LIN {X -0.110,Y -591.077,Z 1525.096,A 0.000,B 0.000,C 90.000,E1 53.336} C_DIS
LIN {X 0.114,Y -591.584,Z 1525.089,A 0.000,B 0.000,C 90.000,E1 51.984} C_DIS
LIN {X 0.039,Y -592.394,Z 1525.077,A 0.000,B 0.000,C 90.000,E1 49.865} C_DIS
LIN {X -0.237,Y -592.697,Z 1525.073,A 0.000,B 0.000,C 90.000,E1 49.094} C_DIS
LIN {X 0.093,Y -592.919,Z 1525.067,A 0.000,B 0.000,C 90.000,E1 48.000} C_DIS
LIN {X 0.028,Y -592.937,Z 1525.061,A 0.000,B 0.000,C 90.000,E1 46.944} C_DIS
LIN {X -0.066,Y -592.710,Z 1525.055,A 0.000,B 0.000,C 90.000,E1 45.891} C_DIS
LIN {X -0.158,Y -592.347,Z 1525.049,A 0.000,B 0.000,C 90.000,E1 44.838} C_DIS
LIN {X -0.256,Y -591.689,Z 1525.043,A 0.000,B 0.000,C 90.000,E1 43.785} C_DIS
LIN {X 0.062,Y -590.876,Z 1525.037,A 0.000,B 0.000,C 90.000,E1 42.690} C_DIS
LIN {X 0.018,Y -590.208,Z 1525.034,A 0.000,B 0.000,C 90.000,E1 42.162} C_DIS
LIN {X -0.026,Y -589.196,Z 1525.031,A 0.000,B 0.000,C 90.000,E1 41.634} C_DIS
LIN {X 0.310,Y -587.829,Z 1525.028,A 0.000,B 0.000,C 90.000,E1 41.067} C_DIS
LIN {X 0.059,Y -587.019,Z 1525.027,A 0.000,B 0.000,C 90.000,E1 40.825} C_DIS
LIN {X -0.293,Y -585.430,Z 1525.025,A 0.000,B 0.000,C 90.000,E1 40.458} C_DIS
LIN {X -0.107,Y -583.916,Z 1525.023,A 0.000,B 0.000,C 90.000,E1 40.172} C_DIS
LIN {X -0.139,Y -582.504,Z 1525.022,A 0.000,B 0.000,C 90.000,E1 40.011} C_DIS
LIN {X -0.060,Y -581.396,Z 1525.022,A 0.000,B 0.000,C 90.000,E1 39.930} C_DIS
LIN {X -0.252,Y -580.763,Z 1525.022,A 0.000,B 0.000,C 90.000,E1 39.930} C_DIS
LIN {X 0.106,Y -408.220,Z 1525.022,A 0.000,B 0.000,C 90.000,E1 39.886} C_DIS
LIN {X -0.052,Y -405.621,Z 1525.013,A 0.000,B 0.000,C 90.000,E1 38.382} C_DIS
LIN {X 0.011,Y -396.780,Z 1524.988,A 0.000,B 0.000,C 90.000,E1 33.833} C_DIS
LIN {X -0.015,Y -393.578,Z 1524.976,A 0.000,B 0.000,C 90.000,E1 31.720} C_DIS
LIN {X -0.106,Y -386.207,Z 1524.953,A 0.000,B 0.000,C 90.000,E1 27.462} C_DIS
LIN {X -0.128,Y -382.999,Z 1524.939,A 0.000,B 0.000,C 90.000,E1 24.951} C_DIS
LIN {X -0.025,Y -380.145,Z 1524.929,A 0.000,B 0.000,C 90.000,E1 23.131} C_DIS
LIN {X -0.152,Y -374.085,Z 1524.900,A 0.000,B 0.000,C 90.000,E1 18.055} C_DIS
LIN {X 0.155,Y -373.383,Z 1524.896,A 0.000,B 0.000,C 90.000,E1 17.275} C_DIS
LIN {X 0.170,Y -367.880,Z 1524.868,A 0.000,B 0.000,C 90.000,E1 12.119} C_DIS
LIN {X 0.114,Y -366.486,Z 1524.855,A 0.000,B 0.000,C 90.000,E1 9.905} C_DIS
LIN {X 0.050,Y -361.788,Z 1524.822,A 0.000,B 0.000,C 90.000,E1 3.955} C_DIS
LIN {X -0.065,Y -360.902,Z 1524.801,A 0.000,B 0.000,C 90.000,E1 0.229} C_DIS
LIN {X -0.053,Y -359.426,Z 1524.770,A 0.000,B 0.000,C 90.000,E1 354.546} C_DIS
LIN {X 0.070,Y -358.890,Z 1524.759,A 0.000,B 0.000,C 90.000,E1 352.648} C_DIS
LIN {X -0.020,Y -359.563,Z 1524.726,A 0.000,B 0.000,C 90.000,E1 346.645} C_DIS
LIN {X 0.001,Y -361.801,Z 1524.684,A 0.000,B 0.000,C 90.000,E1 339.135} C_DIS
LIN {X -0.154,Y -362.053,Z 1524.680,A 0.000,B 0.000,C 90.000,E1 338.411} C_DIS
LIN {X 0.189,Y -365.980,Z 1524.643,A 0.000,B 0.000,C 90.000,E1 331.641} C_DIS
LIN {X 0.029,Y -366.387,Z 1524.639,A 0.000,B 0.000,C 90.000,E1 330.923} C_DIS
LIN {X -0.031,Y -371.355,Z 1524.604,A 0.000,B 0.000,C 90.000,E1 324.642} C_DIS
LIN {X -0.043,Y -371.766,Z 1524.602,A 0.000,B 0.000,C 90.000,E1 324.276} C_DIS
LIN {X 0.013,Y -377.358,Z 1524.567,A 0.000,B 0.000,C 90.000,E1 318.038} C_DIS
LIN {X 0.012,Y -378.235,Z 1524.563,A 0.000,B 0.000,C 90.000,E1 317.310} C_DIS
LIN {X 0.002,Y -383.940,Z 1524.531,A 0.000,B 0.000,C 90.000,E1 311.515} C_DIS
LIN {X 0.088,Y -384.893,Z 1524.527,A 0.000,B 0.000,C 90.000,E1 310.782} C_DIS
LIN {X 0.262,Y -390.610,Z 1524.495,A 0.000,B 0.000,C 90.000,E1 305.025} C_DIS
LIN {X 0.106,Y -391.104,Z 1524.493,A 0.000,B 0.000,C 90.000,E1 304.692} C_DIS
LIN {X 0.022,Y -391.648,Z 1524.489,A 0.000,B 0.000,C 90.000,E1 303.992} C_DIS
LIN {X -0.080,Y -396.825,Z 1524.459,A 0.000,B 0.000,C 90.000,E1 298.693} C_DIS
LIN {X -0.210,Y -397.120,Z 1524.457,A 0.000,B 0.000,C 90.000,E1 298.359} C_DIS
LIN {X -0.055,Y -401.597,Z 1524.426,A 0.000,B 0.000,C 90.000,E1 292.717} C_DIS
LIN {X 0.222,Y -404.659,Z 1524.395,A 0.000,B 0.000,C 90.000,E1 287.094} C_DIS
LIN {X -0.079,Y -404.735,Z 1524.391,A 0.000,B 0.000,C 90.000,E1 286.441} C_DIS
LIN {X 0.214,Y -406.099,Z 1524.364,A 0.000,B 0.000,C 90.000,E1 281.535} C_DIS
LIN {X -0.176,Y -406.094,Z 1524.362,A 0.000,B 0.000,C 90.000,E1 281.243} C_DIS
LIN {X -0.097,Y -405.680,Z 1524.333,A 0.000,B 0.000,C 90.000,E1 276.024} C_DIS
LIN {X -0.165,Y -405.058,Z 1524.328,A 0.000,B 0.000,C 90.000,E1 274.992} C_DIS
LIN {X -0.060,Y -403.497,Z 1524.304,A 0.000,B 0.000,C 90.000,E1 270.802} C_DIS
LIN {X -0.092,Y -403.288,Z 1524.302,A 0.000,B 0.000,C 90.000,E1 270.458} C_DIS
LIN {X 0.091,Y -398.931,Z 1524.271,A 0.000,B 0.000,C 90.000,E1 264.837} C_DIS
LIN {X -0.040,Y -393.108,Z 1524.242,A 0.000,B 0.000,C 90.000,E1 259.567} C_DIS
LIN {X -0.079,Y -392.835,Z 1524.240,A 0.000,B 0.000,C 90.000,E1 259.218} C_DIS
LIN {X 0.034,Y -385.993,Z 1524.212,A 0.000,B 0.000,C 90.000,E1 254.212} C_DIS
LIN {X -0.026,Y -385.267,Z 1524.208,A 0.000,B 0.000,C 90.000,E1 253.504} C_DIS
LIN {X -0.004,Y -384.768,Z 1524.206,A 0.000,B 0.000,C 90.000,E1 253.142} C_DIS
LIN {X 0.221,Y -377.973,Z 1524.182,A 0.000,B 0.000,C 90.000,E1 248.773} C_DIS
LIN {X -0.044,Y -376.233,Z 1524.174,A 0.000,B 0.000,C 90.000,E1 247.358} C_DIS
LIN {X 0.057,Y -374.944,Z 1524.170,A 0.000,B 0.000,C 90.000,E1 246.613} C_DIS
LIN {X -0.208,Y -368.417,Z 1524.148,A 0.000,B 0.000,C 90.000,E1 242.615} C_DIS
LIN {X 0.097,Y -366.047,Z 1524.137,A 0.000,B 0.000,C 90.000,E1 240.717} C_DIS
LIN {X 0.004,Y -359.196,Z 1524.115,A 0.000,B 0.000,C 90.000,E1 236.628} C_DIS
LIN {X 0.021,Y -355.842,Z 1524.100,A 0.000,B 0.000,C 90.000,E1 233.989} C_DIS
LIN {X -0.173,Y -348.793,Z 1524.075,A 0.000,B 0.000,C 90.000,E1 229.461} C_DIS
LIN {X -0.097,Y -346.185,Z 1524.062,A 0.000,B 0.000,C 90.000,E1 227.148} C_DIS
LIN {X -0.088,Y -345.065,Z 1524.058,A 0.000,B 0.000,C 90.000,E1 226.377} C_DIS
LIN {X 0.094,Y -338.586,Z 1524.030,A 0.000,B 0.000,C 90.000,E1 221.310} C_DIS
LIN {X 0.094,Y -336.840,Z 1524.019,A 0.000,B 0.000,C 90.000,E1 219.358} C_DIS
LIN {X 0.014,Y -330.861,Z 1523.988,A 0.000,B 0.000,C 90.000,E1 213.865} C_DIS
LIN {X 0.149,Y -329.296,Z 1523.975,A 0.000,B 0.000,C 90.000,E1 211.465} C_DIS
LIN {X -0.154,Y -324.669,Z 1523.942,A 0.000,B 0.000,C 90.000,E1 205.540} C_DIS
LIN {X 0.174,Y -323.837,Z 1523.928,A 0.000,B 0.000,C 90.000,E1 203.078} C_DIS
LIN {X -0.017,Y -321.124,Z 1523.881,A 0.000,B 0.000,C 90.000,E1 194.662} C_DIS
LIN {X 0.138,Y -320.932,Z 1523.877,A 0.000,B 0.000,C 90.000,E1 193.828} C_DIS
LIN {X -0.076,Y -321.562,Z 1523.832,A 0.000,B 0.000,C 90.000,E1 185.796} C_DIS
LIN {X -0.143,Y -324.415,Z 1523.790,A 0.000,B 0.000,C 90.000,E1 178.165} C_DIS
LIN {X -0.141,Y -325.376,Z 1523.783,A 0.000,B 0.000,C 90.000,E1 176.963} C_DIS
LIN {X -0.100,Y -329.112,Z 1523.750,A 0.000,B 0.000,C 90.000,E1 170.971} C_DIS
LIN {X 0.061,Y -334.260,Z 1523.726,A 0.000,B 0.000,C 90.000,E1 166.589} C_DIS
LIN {X 0.067,Y -335.488,Z 1523.719,A 0.000,B 0.000,C 90.000,E1 165.408} C_DIS
LIN {X 0.143,Y -340.932,Z 1523.695,A 0.000,B 0.000,C 90.000,E1 161.094} C_DIS
LIN {X -0.172,Y -342.138,Z 1523.691,A 0.000,B 0.000,C 90.000,E1 160.369} C_DIS
LIN {X -0.058,Y -347.939,Z 1523.667,A 0.000,B 0.000,C 90.000,E1 156.102} C_DIS
LIN {X -0.081,Y -354.259,Z 1523.648,A 0.000,B 0.000,C 90.000,E1 152.666} C_DIS
LIN {X -0.222,Y -361.406,Z 1523.625,A 0.000,B 0.000,C 90.000,E1 148.535} C_DIS
LIN {X 0.065,Y -368.758,Z 1523.606,A 0.000,B 0.000,C 90.000,E1 145.135} C_DIS
LIN {X 0.065,Y -377.029,Z 1523.584,A 0.000,B 0.000,C 90.000,E1 141.090} C_DIS
LIN {X -0.061,Y -383.435,Z 1523.570,A 0.000,B 0.000,C 90.000,E1 138.566} C_DIS
LIN {X -0.015,Y -385.037,Z 1523.566,A 0.000,B 0.000,C 90.000,E1 137.838} C_DIS
LIN {X -0.132,Y -386.364,Z 1523.562,A 0.000,B 0.000,C 90.000,E1 137.229} C_DIS
LIN {X -0.232,Y -540.923,Z 1523.562,A 0.000,B 0.000,C 90.000,E1 137.229} C_DIS
LIN {X 0.102,Y -542.616,Z 1523.562,A 0.000,B 0.000,C 90.000,E1 137.106} C_DIS
LIN {X -0.112,Y -544.188,Z 1523.561,A 0.000,B 0.000,C 90.000,E1 136.944} C_DIS
LIN {X -0.124,Y -545.786,Z 1523.559,A 0.000,B 0.000,C 90.000,E1 136.662} C_DIS
LIN {X -0.104,Y -546.970,Z 1523.558,A 0.000,B 0.000,C 90.000,E1 136.377} C_DIS
LIN {X -0.074,Y -548.801,Z 1523.555,A 0.000,B 0.000,C 90.000,E1 135.810} C_DIS
LIN {X -0.029,Y -550.156,Z 1523.551,A 0.000,B 0.000,C 90.000,E1 135.243} C_DIS
LIN {X 0.028,Y -551.193,Z 1523.548,A 0.000,B 0.000,C 90.000,E1 134.676} C_DIS
LIN {X -0.264,Y -552.360,Z 1523.544,A 0.000,B 0.000,C 90.000,E1 133.866} C_DIS
LIN {X -0.070,Y -553.654,Z 1523.536,A 0.000,B 0.000,C 90.000,E1 132.447} C_DIS
LIN {X -0.227,Y -554.854,Z 1523.528,A 0.000,B 0.000,C 90.000,E1 131.067} C_DIS
LIN {X 0.058,Y -555.934,Z 1523.520,A 0.000,B 0.000,C 90.000,E1 129.644} C_DIS
LIN {X 0.012,Y -556.872,Z 1523.513,A 0.000,B 0.000,C 90.000,E1 128.257} C_DIS
LIN {X -0.017,Y -557.730,Z 1523.505,A 0.000,B 0.000,C 90.000,E1 126.870} C_DIS
LIN {X 0.321,Y -558.307,Z 1523.499,A 0.000,B 0.000,C 90.000,E1 125.724} C_DIS
LIN {X -0.117,Y -558.754,Z 1523.493,A 0.000,B 0.000,C 90.000,E1 124.659} C_DIS
LIN {X 0.370,Y -559.049,Z 1523.486,A 0.000,B 0.000,C 90.000,E1 123.499} C_DIS
LIN {X 0.176,Y -559.194,Z 1523.479,A 0.000,B 0.000,C 90.000,E1 122.133} C_DIS
LIN {X -0.106,Y -559.571,Z 1523.465,A 0.000,B 0.000,C 90.000,E1 119.667} C_DIS
LIN {X -0.106,Y -559.896,Z 1523.457,A 0.000,B 0.000,C 90.000,E1 118.281} C_DIS
LIN {X 0.128,Y -560.256,Z 1523.449,A 0.000,B 0.000,C 90.000,E1 116.873} C_DIS
LIN {X -0.133,Y -560.520,Z 1523.442,A 0.000,B 0.000,C 90.000,E1 115.515} C_DIS
LIN {X -0.027,Y -560.874,Z 1523.431,A 0.000,B 0.000,C 90.000,E1 113.567} C_DIS
LIN {X -0.240,Y -561.086,Z 1523.423,A 0.000,B 0.000,C 90.000,E1 112.206} C_DIS
LIN {X 0.075,Y -561.325,Z 1523.416,A 0.000,B 0.000,C 90.000,E1 110.791} C_DIS
LIN {X -0.016,Y -561.627,Z 1523.406,A 0.000,B 0.000,C 90.000,E1 109.141} C_DIS
LIN {X 0.246,Y -561.910,Z 1523.397,A 0.000,B 0.000,C 90.000,E1 107.457} C_DIS
LIN {X -0.185,Y -562.229,Z 1523.388,A 0.000,B 0.000,C 90.000,E1 105.843} C_DIS
LIN {X -0.074,Y -562.589,Z 1523.379,A 0.000,B 0.000,C 90.000,E1 104.175} C_DIS
LIN {X -0.229,Y -563.011,Z 1523.370,A 0.000,B 0.000,C 90.000,E1 102.535} C_DIS
LIN {X -0.206,Y -563.703,Z 1523.359,A 0.000,B 0.000,C 90.000,E1 100.602} C_DIS
LIN {X 0.276,Y -564.452,Z 1523.348,A 0.000,B 0.000,C 90.000,E1 98.624} C_DIS
LIN {X -0.196,Y -565.016,Z 1523.340,A 0.000,B 0.000,C 90.000,E1 97.296} C_DIS
LIN {X 0.001,Y -565.710,Z 1523.331,A 0.000,B 0.000,C 90.000,E1 95.625} C_DIS
LIN {X -0.246,Y -566.525,Z 1523.321,A 0.000,B 0.000,C 90.000,E1 93.726} C_DIS
LIN {X -0.095,Y -567.254,Z 1523.311,A 0.000,B 0.000,C 90.000,E1 92.064} C_DIS
LIN {X -0.048,Y -567.928,Z 1523.304,A 0.000,B 0.000,C 90.000,E1 90.688} C_DIS
LIN {X 0.123,Y -568.719,Z 1523.295,A 0.000,B 0.000,C 90.000,E1 89.026} C_DIS
LIN {X 0.031,Y -569.821,Z 1523.283,A 0.000,B 0.000,C 90.000,E1 86.846} C_DIS
LIN {X -0.154,Y -570.797,Z 1523.272,A 0.000,B 0.000,C 90.000,E1 84.951} C_DIS
LIN {X -0.011,Y -571.595,Z 1523.264,A 0.000,B 0.000,C 90.000,E1 83.571} C_DIS
LIN {X 0.022,Y -572.832,Z 1523.254,A 0.000,B 0.000,C 90.000,E1 81.659} C_DIS
LIN {X 0.092,Y -574.108,Z 1523.243,A 0.000,B 0.000,C 90.000,E1 79.746} C_DIS
LIN {X -0.283,Y -575.573,Z 1523.233,A 0.000,B 0.000,C 90.000,E1 77.881} C_DIS
LIN {X -0.026,Y -576.844,Z 1523.224,A 0.000,B 0.000,C 90.000,E1 76.228} C_DIS
LIN {X -0.307,Y -577.653,Z 1523.218,A 0.000,B 0.000,C 90.000,E1 75.172} C_DIS
LIN {X -0.205,Y -578.921,Z 1523.207,A 0.000,B 0.000,C 90.000,E1 73.268} C_DIS
LIN {X -0.075,Y -580.324,Z 1523.195,A 0.000,B 0.000,C 90.000,E1 71.094} C_DIS
LIN {X -0.190,Y -580.822,Z 1523.190,A 0.000,B 0.000,C 90.000,E1 70.296} C_DIS
LIN {X 0.147,Y -581.736,Z 1523.182,A 0.000,B 0.000,C 90.000,E1 68.646} C_DIS
LIN {X -0.185,Y -582.761,Z 1523.171,A 0.000,B 0.000,C 90.000,E1 66.794} C_DIS
LIN {X -0.274,Y -583.826,Z 1523.161,A 0.000,B 0.000,C 90.000,E1 64.921} C_DIS
LIN {X -0.213,Y -585.515,Z 1523.146,A 0.000,B 0.000,C 90.000,E1 62.231} C_DIS
LIN {X 0.137,Y -586.676,Z 1523.137,A 0.000,B 0.000,C 90.000,E1 60.589} C_DIS
LIN {X -0.175,Y -587.630,Z 1523.129,A 0.000,B 0.000,C 90.000,E1 59.282} C_DIS
LIN {X 0.134,Y -588.545,Z 1523.122,A 0.000,B 0.000,C 90.000,E1 57.916} C_DIS
LIN {X 0.146,Y -589.451,Z 1523.115,A 0.000,B 0.000,C 90.000,E1 56.580} C_DIS
LIN {X -0.003,Y -590.403,Z 1523.107,A 0.000,B 0.000,C 90.000,E1 55.261} C_DIS
LIN {X -0.199,Y -591.398,Z 1523.097,A 0.000,B 0.000,C 90.000,E1 53.417} C_DIS
LIN {X 0.028,Y -591.926,Z 1523.089,A 0.000,B 0.000,C 90.000,E1 52.065} C_DIS
LIN {X 0.342,Y -592.766,Z 1523.078,A 0.000,B 0.000,C 90.000,E1 49.908} C_DIS
LIN {X 0.283,Y -593.108,Z 1523.072,A 0.000,B 0.000,C 90.000,E1 48.852} C_DIS
LIN {X 0.020,Y -593.337,Z 1523.067,A 0.000,B 0.000,C 90.000,E1 48.081} C_DIS
LIN {X -0.039,Y -593.355,Z 1523.061,A 0.000,B 0.000,C 90.000,E1 47.025} C_DIS
LIN {X -0.359,Y -593.143,Z 1523.054,A 0.000,B 0.000,C 90.000,E1 45.729} C_DIS
LIN {X -0.029,Y -592.727,Z 1523.048,A 0.000,B 0.000,C 90.000,E1 44.636} C_DIS
LIN {X 0.061,Y -591.812,Z 1523.041,A 0.000,B 0.000,C 90.000,E1 43.299} C_DIS
LIN {X -0.019,Y -590.948,Z 1523.035,A 0.000,B 0.000,C 90.000,E1 42.243} C_DIS
LIN {X 0.090,Y -589.887,Z 1523.030,A 0.000,B 0.000,C 90.000,E1 41.434} C_DIS
LIN {X 0.040,Y -588.904,Z 1523.027,A 0.000,B 0.000,C 90.000,E1 40.906} C_DIS
LIN {X -0.016,Y -587.630,Z 1523.024,A 0.000,B 0.000,C 90.000,E1 40.378} C_DIS
LIN {X 0.177,Y -586.831,Z 1523.023,A 0.000,B 0.000,C 90.000,E1 40.092} C_DIS
LIN {X -0.080,Y -585.891,Z 1523.021,A 0.000,B 0.000,C 90.000,E1 39.850} C_DIS
LIN {X 0.109,Y -584.616,Z 1523.020,A 0.000,B 0.000,C 90.000,E1 39.564} C_DIS
LIN {X 0.016,Y -583.816,Z 1523.019,A 0.000,B 0.000,C 90.000,E1 39.439} C_DIS
LIN {X -0.294,Y -582.284,Z 1523.018,A 0.000,B 0.000,C 90.000,E1 39.277} C_DIS
LIN {X -0.299,Y -581.245,Z 1523.018,A 0.000,B 0.000,C 90.000,E1 39.197} C_DIS
LIN {X 0.095,Y -580.125,Z 1523.017,A 0.000,B 0.000,C 90.000,E1 39.116} C_DIS
LIN {X 0.043,Y -406.894,Z 1523.017,A 0.000,B 0.000,C 90.000,E1 39.116} C_DIS
LIN {X 0.050,Y -405.552,Z 1523.013,A 0.000,B 0.000,C 90.000,E1 38.338} C_DIS
LIN {X 0.125,Y -396.729,Z 1522.988,A 0.000,B 0.000,C 90.000,E1 33.785} C_DIS
LIN {X 0.105,Y -393.515,Z 1522.976,A 0.000,B 0.000,C 90.000,E1 31.671} C_DIS
LIN {X 0.200,Y -386.161,Z 1522.952,A 0.000,B 0.000,C 90.000,E1 27.385} C_DIS
LIN {X 0.006,Y -382.963,Z 1522.938,A 0.000,B 0.000,C 90.000,E1 24.899} C_DIS
LIN {X 0.104,Y -376.256,Z 1522.912,A 0.000,B 0.000,C 90.000,E1 20.174} C_DIS
LIN {X -0.031,Y -373.747,Z 1522.898,A 0.000,B 0.000,C 90.000,E1 17.638} C_DIS
LIN {X -0.112,Y -372.359,Z 1522.892,A 0.000,B 0.000,C 90.000,E1 16.551} C_DIS
LIN {X -0.030,Y -367.091,Z 1522.861,A 0.000,B 0.000,C 90.000,E1 11.007} C_DIS
LIN {X -0.096,Y -366.466,Z 1522.855,A 0.000,B 0.000,C 90.000,E1 9.905} C_DIS
LIN {X -0.158,Y -361.773,Z 1522.822,A 0.000,B 0.000,C 90.000,E1 3.955} C_DIS
LIN {X 0.088,Y -360.895,Z 1522.801,A 0.000,B 0.000,C 90.000,E1 0.172} C_DIS
LIN {X -0.053,Y -359.426,Z 1522.770,A 0.000,B 0.000,C 90.000,E1 354.546} C_DIS
LIN {X 0.070,Y -358.890,Z 1522.759,A 0.000,B 0.000,C 90.000,E1 352.648} C_DIS
LIN {X -0.020,Y -359.563,Z 1522.726,A 0.000,B 0.000,C 90.000,E1 346.645} C_DIS
LIN {X 0.001,Y -361.801,Z 1522.684,A 0.000,B 0.000,C 90.000,E1 339.135} C_DIS
LIN {X -0.154,Y -362.053,Z 1522.680,A 0.000,B 0.000,C 90.000,E1 338.411} C_DIS
LIN {X 0.189,Y -365.980,Z 1522.643,A 0.000,B 0.000,C 90.000,E1 331.641} C_DIS
LIN {X 0.029,Y -366.387,Z 1522.639,A 0.000,B 0.000,C 90.000,E1 330.923} C_DIS
LIN {X -0.031,Y -371.355,Z 1522.604,A 0.000,B 0.000,C 90.000,E1 324.642} C_DIS
LIN {X -0.043,Y -371.766,Z 1522.602,A 0.000,B 0.000,C 90.000,E1 324.276} C_DIS
LIN {X 0.013,Y -377.358,Z 1522.567,A 0.000,B 0.000,C 90.000,E1 318.038} C_DIS
LIN {X 0.012,Y -378.235,Z 1522.563,A 0.000,B 0.000,C 90.000,E1 317.310} C_DIS
LIN {X 0.002,Y -383.940,Z 1522.531,A 0.000,B 0.000,C 90.000,E1 311.515} C_DIS
LIN {X 0.088,Y -384.893,Z 1522.527,A 0.000,B 0.000,C 90.000,E1 310.782} C_DIS
LIN {X 0.262,Y -390.610,Z 1522.495,A 0.000,B 0.000,C 90.000,E1 305.025} C_DIS
LIN {X 0.106,Y -391.104,Z 1522.493,A 0.000,B 0.000,C 90.000,E1 304.692} C_DIS
LIN {X 0.022,Y -391.648,Z 1522.489,A 0.000,B 0.000,C 90.000,E1 303.992} C_DIS
LIN {X -0.080,Y -396.825,Z 1522.459,A 0.000,B 0.000,C 90.000,E1 298.693} C_DIS
LIN {X -0.210,Y -397.120,Z 1522.457,A 0.000,B 0.000,C 90.000,E1 298.359} C_DIS
LIN {X -0.055,Y -401.597,Z 1522.426,A 0.000,B 0.000,C 90.000,E1 292.717} C_DIS
LIN {X 0.222,Y -404.659,Z 1522.395,A 0.000,B 0.000,C 90.000,E1 287.094} C_DIS
LIN {X -0.079,Y -404.735,Z 1522.391,A 0.000,B 0.000,C 90.000,E1 286.441} C_DIS
LIN {X 0.214,Y -406.099,Z 1522.364,A 0.000,B 0.000,C 90.000,E1 281.535} C_DIS
LIN {X -0.176,Y -406.094,Z 1522.362,A 0.000,B 0.000,C 90.000,E1 281.243} C_DIS
LIN {X -0.097,Y -405.680,Z 1522.333,A 0.000,B 0.000,C 90.000,E1 276.024} C_DIS
LIN {X -0.165,Y -405.058,Z 1522.328,A 0.000,B 0.000,C 90.000,E1 274.992} C_DIS
LIN {X -0.060,Y -403.497,Z 1522.304,A 0.000,B 0.000,C 90.000,E1 270.802} C_DIS
LIN {X -0.092,Y -403.288,Z 1522.302,A 0.000,B 0.000,C 90.000,E1 270.458} C_DIS
LIN {X 0.091,Y -398.931,Z 1522.271,A 0.000,B 0.000,C 90.000,E1 264.837} C_DIS
LIN {X -0.040,Y -393.108,Z 1522.242,A 0.000,B 0.000,C 90.000,E1 259.567} C_DIS
LIN {X -0.079,Y -392.835,Z 1522.240,A 0.000,B 0.000,C 90.000,E1 259.218} C_DIS
LIN {X 0.034,Y -385.993,Z 1522.212,A 0.000,B 0.000,C 90.000,E1 254.212} C_DIS
LIN {X -0.026,Y -385.267,Z 1522.208,A 0.000,B 0.000,C 90.000,E1 253.504} C_DIS
LIN {X -0.004,Y -384.768,Z 1522.206,A 0.000,B 0.000,C 90.000,E1 253.142} C_DIS
LIN {X 0.221,Y -377.973,Z 1522.182,A 0.000,B 0.000,C 90.000,E1 248.773} C_DIS
LIN {X -0.044,Y -376.233,Z 1522.174,A 0.000,B 0.000,C 90.000,E1 247.358} C_DIS
LIN {X 0.057,Y -374.944,Z 1522.170,A 0.000,B 0.000,C 90.000,E1 246.613} C_DIS
LIN {X -0.208,Y -368.417,Z 1522.148,A 0.000,B 0.000,C 90.000,E1 242.615} C_DIS
LIN {X 0.097,Y -366.047,Z 1522.137,A 0.000,B 0.000,C 90.000,E1 240.717} C_DIS
LIN {X 0.004,Y -359.196,Z 1522.115,A 0.000,B 0.000,C 90.000,E1 236.628} C_DIS
LIN {X 0.021,Y -355.842,Z 1522.100,A 0.000,B 0.000,C 90.000,E1 233.989} C_DIS
LIN {X -0.173,Y -348.793,Z 1522.075,A 0.000,B 0.000,C 90.000,E1 229.461} C_DIS
LIN {X -0.097,Y -346.185,Z 1522.062,A 0.000,B 0.000,C 90.000,E1 227.148} C_DIS
LIN {X -0.088,Y -345.065,Z 1522.058,A 0.000,B 0.000,C 90.000,E1 226.377} C_DIS
LIN {X 0.094,Y -338.586,Z 1522.030,A 0.000,B 0.000,C 90.000,E1 221.310} C_DIS
LIN {X 0.094,Y -336.840,Z 1522.019,A 0.000,B 0.000,C 90.000,E1 219.358} C_DIS
LIN {X 0.014,Y -330.861,Z 1521.988,A 0.000,B 0.000,C 90.000,E1 213.865} C_DIS
LIN {X 0.149,Y -329.296,Z 1521.975,A 0.000,B 0.000,C 90.000,E1 211.465} C_DIS
LIN {X -0.154,Y -324.669,Z 1521.942,A 0.000,B 0.000,C 90.000,E1 205.540} C_DIS
LIN {X 0.174,Y -323.837,Z 1521.928,A 0.000,B 0.000,C 90.000,E1 203.078} C_DIS
LIN {X -0.017,Y -321.124,Z 1521.881,A 0.000,B 0.000,C 90.000,E1 194.662} C_DIS
LIN {X 0.138,Y -320.932,Z 1521.877,A 0.000,B 0.000,C 90.000,E1 193.828} C_DIS
LIN {X -0.076,Y -321.562,Z 1521.832,A 0.000,B 0.000,C 90.000,E1 185.796} C_DIS
LIN {X -0.143,Y -324.415,Z 1521.790,A 0.000,B 0.000,C 90.000,E1 178.165} C_DIS
LIN {X -0.141,Y -325.376,Z 1521.783,A 0.000,B 0.000,C 90.000,E1 176.963} C_DIS
LIN {X -0.100,Y -329.112,Z 1521.750,A 0.000,B 0.000,C 90.000,E1 170.971} C_DIS
LIN {X 0.061,Y -334.260,Z 1521.726,A 0.000,B 0.000,C 90.000,E1 166.589} C_DIS
LIN {X 0.067,Y -335.488,Z 1521.719,A 0.000,B 0.000,C 90.000,E1 165.408} C_DIS
LIN {X 0.143,Y -340.932,Z 1521.695,A 0.000,B 0.000,C 90.000,E1 161.094} C_DIS
LIN {X -0.172,Y -342.138,Z 1521.691,A 0.000,B 0.000,C 90.000,E1 160.369} C_DIS
LIN {X -0.058,Y -347.939,Z 1521.667,A 0.000,B 0.000,C 90.000,E1 156.102} C_DIS
LIN {X -0.081,Y -354.259,Z 1521.648,A 0.000,B 0.000,C 90.000,E1 152.666} C_DIS
LIN {X -0.222,Y -361.406,Z 1521.625,A 0.000,B 0.000,C 90.000,E1 148.535} C_DIS
LIN {X 0.065,Y -368.758,Z 1521.606,A 0.000,B 0.000,C 90.000,E1 145.135} C_DIS
LIN {X 0.065,Y -377.029,Z 1521.584,A 0.000,B 0.000,C 90.000,E1 141.090} C_DIS
LIN {X -0.061,Y -383.435,Z 1521.570,A 0.000,B 0.000,C 90.000,E1 138.566} C_DIS
LIN {X -0.153,Y -384.579,Z 1521.567,A 0.000,B 0.000,C 90.000,E1 138.081} C_DIS
LIN {X -0.249,Y -540.182,Z 1521.567,A 0.000,B 0.000,C 90.000,E1 138.081} C_DIS
LIN {X 0.231,Y -542.118,Z 1521.566,A 0.000,B 0.000,C 90.000,E1 137.919} C_DIS
LIN {X -0.021,Y -543.063,Z 1521.566,A 0.000,B 0.000,C 90.000,E1 137.838} C_DIS
LIN {X -0.196,Y -544.018,Z 1521.565,A 0.000,B 0.000,C 90.000,E1 137.715} C_DIS
LIN {X 0.190,Y -545.485,Z 1521.563,A 0.000,B 0.000,C 90.000,E1 137.391} C_DIS
LIN {X 0.010,Y -547.099,Z 1521.561,A 0.000,B 0.000,C 90.000,E1 136.986} C_DIS
LIN {X 0.042,Y -548.741,Z 1521.558,A 0.000,B 0.000,C 90.000,E1 136.419} C_DIS
LIN {X -0.293,Y -550.004,Z 1521.555,A 0.000,B 0.000,C 90.000,E1 135.891} C_DIS
LIN {X -0.239,Y -550.989,Z 1521.552,A 0.000,B 0.000,C 90.000,E1 135.324} C_DIS
LIN {X 0.248,Y -552.037,Z 1521.547,A 0.000,B 0.000,C 90.000,E1 134.433} C_DIS
LIN {X -0.035,Y -552.923,Z 1521.542,A 0.000,B 0.000,C 90.000,E1 133.623} C_DIS
LIN {X 0.168,Y -554.208,Z 1521.535,A 0.000,B 0.000,C 90.000,E1 132.204} C_DIS
LIN {X 0.017,Y -555.349,Z 1521.527,A 0.000,B 0.000,C 90.000,E1 130.825} C_DIS
LIN {X -0.122,Y -556.209,Z 1521.521,A 0.000,B 0.000,C 90.000,E1 129.725} C_DIS
LIN {X 0.265,Y -557.294,Z 1521.511,A 0.000,B 0.000,C 90.000,E1 128.016} C_DIS
LIN {X -0.099,Y -558.114,Z 1521.504,A 0.000,B 0.000,C 90.000,E1 126.664} C_DIS
LIN {X 0.247,Y -558.649,Z 1521.498,A 0.000,B 0.000,C 90.000,E1 125.518} C_DIS
LIN {X 0.360,Y -559.144,Z 1521.490,A 0.000,B 0.000,C 90.000,E1 124.119} C_DIS
LIN {X 0.083,Y -559.329,Z 1521.484,A 0.000,B 0.000,C 90.000,E1 123.038} C_DIS
LIN {X -0.102,Y -559.376,Z 1521.476,A 0.000,B 0.000,C 90.000,E1 121.671} C_DIS
LIN {X 0.115,Y -559.816,Z 1521.462,A 0.000,B 0.000,C 90.000,E1 119.155} C_DIS
LIN {X -0.081,Y -560.211,Z 1521.453,A 0.000,B 0.000,C 90.000,E1 117.513} C_DIS
LIN {X -0.138,Y -560.473,Z 1521.447,A 0.000,B 0.000,C 90.000,E1 116.411} C_DIS
LIN {X 0.173,Y -560.756,Z 1521.438,A 0.000,B 0.000,C 90.000,E1 114.719} C_DIS
LIN {X -0.014,Y -561.098,Z 1521.428,A 0.000,B 0.000,C 90.000,E1 113.078} C_DIS
LIN {X -0.114,Y -561.421,Z 1521.417,A 0.000,B 0.000,C 90.000,E1 111.153} C_DIS
LIN {X -0.081,Y -561.731,Z 1521.407,A 0.000,B 0.000,C 90.000,E1 109.214} C_DIS
LIN {X -0.342,Y -562.018,Z 1521.398,A 0.000,B 0.000,C 90.000,E1 107.583} C_DIS
LIN {X -0.070,Y -562.339,Z 1521.388,A 0.000,B 0.000,C 90.000,E1 105.898} C_DIS
LIN {X -0.254,Y -562.667,Z 1521.381,A 0.000,B 0.000,C 90.000,E1 104.537} C_DIS
LIN {X -0.118,Y -563.156,Z 1521.370,A 0.000,B 0.000,C 90.000,E1 102.591} C_DIS
LIN {X 0.066,Y -563.933,Z 1521.358,A 0.000,B 0.000,C 90.000,E1 100.366} C_DIS
LIN {X 0.070,Y -564.861,Z 1521.345,A 0.000,B 0.000,C 90.000,E1 98.163} C_DIS
LIN {X -0.235,Y -565.506,Z 1521.336,A 0.000,B 0.000,C 90.000,E1 96.543} C_DIS
LIN {X -0.190,Y -566.084,Z 1521.329,A 0.000,B 0.000,C 90.000,E1 95.163} C_DIS
LIN {X -0.129,Y -566.724,Z 1521.321,A 0.000,B 0.000,C 90.000,E1 93.784} C_DIS
LIN {X 0.145,Y -567.588,Z 1521.310,A 0.000,B 0.000,C 90.000,E1 91.835} C_DIS
LIN {X 0.199,Y -568.277,Z 1521.303,A 0.000,B 0.000,C 90.000,E1 90.458} C_DIS
LIN {X -0.191,Y -569.093,Z 1521.294,A 0.000,B 0.000,C 90.000,E1 88.854} C_DIS
LIN {X 0.137,Y -570.094,Z 1521.283,A 0.000,B 0.000,C 90.000,E1 86.906} C_DIS
LIN {X -0.010,Y -571.088,Z 1521.272,A 0.000,B 0.000,C 90.000,E1 85.008} C_DIS
LIN {X 0.141,Y -571.885,Z 1521.265,A 0.000,B 0.000,C 90.000,E1 83.628} C_DIS
LIN {X 0.100,Y -573.123,Z 1521.254,A 0.000,B 0.000,C 90.000,E1 81.724} C_DIS
LIN {X 0.264,Y -574.398,Z 1521.244,A 0.000,B 0.000,C 90.000,E1 79.803} C_DIS
LIN {X 0.256,Y -575.625,Z 1521.234,A 0.000,B 0.000,C 90.000,E1 78.173} C_DIS
LIN {X -0.180,Y -576.906,Z 1521.225,A 0.000,B 0.000,C 90.000,E1 76.589} C_DIS
LIN {X -0.107,Y -577.940,Z 1521.218,A 0.000,B 0.000,C 90.000,E1 75.227} C_DIS
LIN {X -0.202,Y -579.007,Z 1521.209,A 0.000,B 0.000,C 90.000,E1 73.614} C_DIS
LIN {X 0.072,Y -579.861,Z 1521.201,A 0.000,B 0.000,C 90.000,E1 72.236} C_DIS
LIN {X -0.154,Y -581.121,Z 1521.191,A 0.000,B 0.000,C 90.000,E1 70.369} C_DIS
LIN {X 0.037,Y -582.156,Z 1521.180,A 0.000,B 0.000,C 90.000,E1 68.465} C_DIS
LIN {X -0.289,Y -583.194,Z 1521.170,A 0.000,B 0.000,C 90.000,E1 66.613} C_DIS
LIN {X -0.127,Y -584.250,Z 1521.160,A 0.000,B 0.000,C 90.000,E1 64.717} C_DIS
LIN {X -0.038,Y -585.986,Z 1521.145,A 0.000,B 0.000,C 90.000,E1 62.025} C_DIS
LIN {X 0.160,Y -586.994,Z 1521.137,A 0.000,B 0.000,C 90.000,E1 60.667} C_DIS
LIN {X 0.029,Y -588.093,Z 1521.128,A 0.000,B 0.000,C 90.000,E1 59.076} C_DIS
LIN {X 0.035,Y -589.004,Z 1521.121,A 0.000,B 0.000,C 90.000,E1 57.740} C_DIS
LIN {X -0.122,Y -589.906,Z 1521.113,A 0.000,B 0.000,C 90.000,E1 56.421} C_DIS
LIN {X -0.256,Y -590.868,Z 1521.106,A 0.000,B 0.000,C 90.000,E1 55.102} C_DIS
LIN {X -0.170,Y -591.696,Z 1521.097,A 0.000,B 0.000,C 90.000,E1 53.497} C_DIS
LIN {X 0.060,Y -592.261,Z 1521.090,A 0.000,B 0.000,C 90.000,E1 52.145} C_DIS
LIN {X -0.047,Y -592.871,Z 1521.081,A 0.000,B 0.000,C 90.000,E1 50.561} C_DIS
LIN {X 0.326,Y -593.519,Z 1521.072,A 0.000,B 0.000,C 90.000,E1 48.933} C_DIS
LIN {X -0.167,Y -593.738,Z 1521.066,A 0.000,B 0.000,C 90.000,E1 47.919} C_DIS
LIN {X 0.186,Y -593.735,Z 1521.060,A 0.000,B 0.000,C 90.000,E1 46.824} C_DIS
LIN {X 0.306,Y -593.535,Z 1521.053,A 0.000,B 0.000,C 90.000,E1 45.486} C_DIS
LIN {X 0.225,Y -593.037,Z 1521.047,A 0.000,B 0.000,C 90.000,E1 44.433} C_DIS
LIN {X 0.134,Y -592.349,Z 1521.041,A 0.000,B 0.000,C 90.000,E1 43.380} C_DIS
LIN {X 0.060,Y -591.464,Z 1521.035,A 0.000,B 0.000,C 90.000,E1 42.324} C_DIS
LIN {X -0.069,Y -590.277,Z 1521.029,A 0.000,B 0.000,C 90.000,E1 41.272} C_DIS
LIN {X -0.117,Y -589.582,Z 1521.026,A 0.000,B 0.000,C 90.000,E1 40.744} C_DIS
LIN {X 0.280,Y -588.642,Z 1521.023,A 0.000,B 0.000,C 90.000,E1 40.172} C_DIS
LIN {X 0.027,Y -588.080,Z 1521.022,A 0.000,B 0.000,C 90.000,E1 39.930} C_DIS
LIN {X 0.224,Y -587.372,Z 1521.020,A 0.000,B 0.000,C 90.000,E1 39.644} C_DIS
LIN {X -0.035,Y -586.521,Z 1521.019,A 0.000,B 0.000,C 90.000,E1 39.402} C_DIS
LIN {X 0.157,Y -585.537,Z 1521.017,A 0.000,B 0.000,C 90.000,E1 39.116} C_DIS
LIN {X 0.346,Y -584.347,Z 1521.016,A 0.000,B 0.000,C 90.000,E1 38.830} C_DIS
LIN {X -0.198,Y -583.596,Z 1521.015,A 0.000,B 0.000,C 90.000,E1 38.749} C_DIS
LIN {X -0.053,Y -582.185,Z 1521.014,A 0.000,B 0.000,C 90.000,E1 38.543} C_DIS
LIN {X -0.345,Y -580.988,Z 1521.014,A 0.000,B 0.000,C 90.000,E1 38.463} C_DIS
LIN {X -0.073,Y -579.954,Z 1521.013,A 0.000,B 0.000,C 90.000,E1 38.382} C_DIS
LIN {X -0.209,Y -579.391,Z 1521.013,A 0.000,B 0.000,C 90.000,E1 38.382} C_DIS
LIN {X -0.170,Y -405.584,Z 1521.013,A 0.000,B 0.000,C 90.000,E1 38.382} C_DIS
LIN {X 0.125,Y -397.278,Z 1520.990,A 0.000,B 0.000,C 90.000,E1 34.119} C_DIS
LIN {X 0.115,Y -394.054,Z 1520.978,A 0.000,B 0.000,C 90.000,E1 32.005} C_DIS
LIN {X -0.019,Y -393.478,Z 1520.976,A 0.000,B 0.000,C 90.000,E1 31.671} C_DIS
LIN {X 0.077,Y -386.135,Z 1520.952,A 0.000,B 0.000,C 90.000,E1 27.385} C_DIS
LIN {X -0.117,Y -382.943,Z 1520.938,A 0.000,B 0.000,C 90.000,E1 24.899} C_DIS
LIN {X -0.018,Y -376.235,Z 1520.912,A 0.000,B 0.000,C 90.000,E1 20.174} C_DIS
LIN {X -0.153,Y -373.731,Z 1520.898,A 0.000,B 0.000,C 90.000,E1 17.638} C_DIS
LIN {X 0.091,Y -371.871,Z 1520.890,A 0.000,B 0.000,C 90.000,E1 16.134} C_DIS
LIN {X 0.068,Y -366.857,Z 1520.859,A 0.000,B 0.000,C 90.000,E1 10.602} C_DIS
LIN {X 0.145,Y -366.452,Z 1520.855,A 0.000,B 0.000,C 90.000,E1 9.849} C_DIS
LIN {X 0.082,Y -361.764,Z 1520.822,A 0.000,B 0.000,C 90.000,E1 3.898} C_DIS
LIN {X -0.033,Y -360.889,Z 1520.801,A 0.000,B 0.000,C 90.000,E1 0.172} C_DIS
LIN {X -0.053,Y -359.426,Z 1520.770,A 0.000,B 0.000,C 90.000,E1 354.546} C_DIS
LIN {X 0.070,Y -358.890,Z 1520.759,A 0.000,B 0.000,C 90.000,E1 352.648} C_DIS
LIN {X -0.020,Y -359.563,Z 1520.726,A 0.000,B 0.000,C 90.000,E1 346.645} C_DIS
LIN {X 0.001,Y -361.801,Z 1520.684,A 0.000,B 0.000,C 90.000,E1 339.135} C_DIS
LIN {X -0.154,Y -362.053,Z 1520.680,A 0.000,B 0.000,C 90.000,E1 338.411} C_DIS
LIN {X 0.189,Y -365.980,Z 1520.643,A 0.000,B 0.000,C 90.000,E1 331.641} C_DIS
LIN {X 0.029,Y -366.387,Z 1520.639,A 0.000,B 0.000,C 90.000,E1 330.923} C_DIS
LIN {X -0.031,Y -371.355,Z 1520.604,A 0.000,B 0.000,C 90.000,E1 324.642} C_DIS
LIN {X -0.043,Y -371.766,Z 1520.602,A 0.000,B 0.000,C 90.000,E1 324.276} C_DIS
LIN {X 0.013,Y -377.358,Z 1520.567,A 0.000,B 0.000,C 90.000,E1 318.038} C_DIS
LIN {X 0.012,Y -378.235,Z 1520.563,A 0.000,B 0.000,C 90.000,E1 317.310} C_DIS
LIN {X 0.002,Y -383.940,Z 1520.531,A 0.000,B 0.000,C 90.000,E1 311.515} C_DIS
LIN {X 0.088,Y -384.893,Z 1520.527,A 0.000,B 0.000,C 90.000,E1 310.782} C_DIS
LIN {X 0.262,Y -390.610,Z 1520.495,A 0.000,B 0.000,C 90.000,E1 305.025} C_DIS
LIN {X 0.106,Y -391.104,Z 1520.493,A 0.000,B 0.000,C 90.000,E1 304.692} C_DIS
LIN {X 0.022,Y -391.648,Z 1520.489,A 0.000,B 0.000,C 90.000,E1 303.992} C_DIS
LIN {X -0.080,Y -396.825,Z 1520.459,A 0.000,B 0.000,C 90.000,E1 298.693} C_DIS
LIN {X -0.210,Y -397.120,Z 1520.457,A 0.000,B 0.000,C 90.000,E1 298.359} C_DIS
LIN {X -0.055,Y -401.597,Z 1520.426,A 0.000,B 0.000,C 90.000,E1 292.717} C_DIS
LIN {X 0.222,Y -404.659,Z 1520.395,A 0.000,B 0.000,C 90.000,E1 287.094} C_DIS
LIN {X -0.079,Y -404.735,Z 1520.391,A 0.000,B 0.000,C 90.000,E1 286.441} C_DIS
LIN {X 0.214,Y -406.099,Z 1520.364,A 0.000,B 0.000,C 90.000,E1 281.535} C_DIS
LIN {X -0.176,Y -406.094,Z 1520.362,A 0.000,B 0.000,C 90.000,E1 281.243} C_DIS
LIN {X -0.097,Y -405.680,Z 1520.333,A 0.000,B 0.000,C 90.000,E1 276.024} C_DIS
LIN {X -0.165,Y -405.058,Z 1520.328,A 0.000,B 0.000,C 90.000,E1 274.992} C_DIS
LIN {X -0.060,Y -403.497,Z 1520.304,A 0.000,B 0.000,C 90.000,E1 270.802} C_DIS
LIN {X -0.092,Y -403.288,Z 1520.302,A 0.000,B 0.000,C 90.000,E1 270.458} C_DIS
LIN {X 0.091,Y -398.931,Z 1520.271,A 0.000,B 0.000,C 90.000,E1 264.837} C_DIS
LIN {X -0.040,Y -393.108,Z 1520.242,A 0.000,B 0.000,C 90.000,E1 259.567} C_DIS
LIN {X -0.079,Y -392.835,Z 1520.240,A 0.000,B 0.000,C 90.000,E1 259.218} C_DIS
LIN {X 0.034,Y -385.993,Z 1520.212,A 0.000,B 0.000,C 90.000,E1 254.212} C_DIS
LIN {X -0.026,Y -385.267,Z 1520.208,A 0.000,B 0.000,C 90.000,E1 253.504} C_DIS
LIN {X -0.004,Y -384.768,Z 1520.206,A 0.000,B 0.000,C 90.000,E1 253.142} C_DIS
LIN {X 0.221,Y -377.973,Z 1520.182,A 0.000,B 0.000,C 90.000,E1 248.773} C_DIS
LIN {X -0.044,Y -376.233,Z 1520.174,A 0.000,B 0.000,C 90.000,E1 247.358} C_DIS
LIN {X 0.057,Y -374.944,Z 1520.170,A 0.000,B 0.000,C 90.000,E1 246.613} C_DIS
LIN {X -0.208,Y -368.417,Z 1520.148,A 0.000,B 0.000,C 90.000,E1 242.615} C_DIS
LIN {X 0.097,Y -366.047,Z 1520.137,A 0.000,B 0.000,C 90.000,E1 240.717} C_DIS
LIN {X 0.004,Y -359.196,Z 1520.115,A 0.000,B 0.000,C 90.000,E1 236.628} C_DIS
LIN {X 0.021,Y -355.842,Z 1520.100,A 0.000,B 0.000,C 90.000,E1 233.989} C_DIS
LIN {X -0.173,Y -348.793,Z 1520.075,A 0.000,B 0.000,C 90.000,E1 229.461} C_DIS
LIN {X -0.097,Y -346.185,Z 1520.062,A 0.000,B 0.000,C 90.000,E1 227.148} C_DIS
LIN {X -0.088,Y -345.065,Z 1520.058,A 0.000,B 0.000,C 90.000,E1 226.377} C_DIS
LIN {X 0.094,Y -338.586,Z 1520.030,A 0.000,B 0.000,C 90.000,E1 221.310} C_DIS
LIN {X 0.094,Y -336.840,Z 1520.019,A 0.000,B 0.000,C 90.000,E1 219.358} C_DIS
LIN {X 0.014,Y -330.861,Z 1519.988,A 0.000,B 0.000,C 90.000,E1 213.865} C_DIS
LIN {X 0.149,Y -329.296,Z 1519.975,A 0.000,B 0.000,C 90.000,E1 211.465} C_DIS
LIN {X -0.154,Y -324.669,Z 1519.942,A 0.000,B 0.000,C 90.000,E1 205.540} C_DIS
LIN {X 0.174,Y -323.837,Z 1519.928,A 0.000,B 0.000,C 90.000,E1 203.078} C_DIS
LIN {X -0.017,Y -321.124,Z 1519.881,A 0.000,B 0.000,C 90.000,E1 194.662} C_DIS
LIN {X 0.138,Y -320.932,Z 1519.877,A 0.000,B 0.000,C 90.000,E1 193.828} C_DIS
LIN {X -0.076,Y -321.562,Z 1519.832,A 0.000,B 0.000,C 90.000,E1 185.796} C_DIS
LIN {X -0.143,Y -324.415,Z 1519.790,A 0.000,B 0.000,C 90.000,E1 178.165} C_DIS
LIN {X -0.141,Y -325.376,Z 1519.783,A 0.000,B 0.000,C 90.000,E1 176.963} C_DIS
LIN {X -0.100,Y -329.112,Z 1519.750,A 0.000,B 0.000,C 90.000,E1 170.971} C_DIS
LIN {X 0.061,Y -334.260,Z 1519.726,A 0.000,B 0.000,C 90.000,E1 166.589} C_DIS
LIN {X 0.067,Y -335.488,Z 1519.719,A 0.000,B 0.000,C 90.000,E1 165.408} C_DIS
LIN {X 0.143,Y -340.932,Z 1519.695,A 0.000,B 0.000,C 90.000,E1 161.094} C_DIS
LIN {X -0.172,Y -342.138,Z 1519.691,A 0.000,B 0.000,C 90.000,E1 160.369} C_DIS
LIN {X -0.058,Y -347.939,Z 1519.667,A 0.000,B 0.000,C 90.000,E1 156.102} C_DIS
LIN {X -0.081,Y -354.259,Z 1519.648,A 0.000,B 0.000,C 90.000,E1 152.666} C_DIS
LIN {X -0.222,Y -361.406,Z 1519.625,A 0.000,B 0.000,C 90.000,E1 148.535} C_DIS
LIN {X 0.065,Y -368.758,Z 1519.606,A 0.000,B 0.000,C 90.000,E1 145.135} C_DIS
LIN {X 0.065,Y -377.029,Z 1519.584,A 0.000,B 0.000,C 90.000,E1 141.090} C_DIS
LIN {X -0.241,Y -382.523,Z 1519.572,A 0.000,B 0.000,C 90.000,E1 138.933} C_DIS
LIN {X -0.035,Y -539.199,Z 1519.572,A 0.000,B 0.000,C 90.000,E1 138.895} C_DIS
LIN {X 0.224,Y -539.838,Z 1519.572,A 0.000,B 0.000,C 90.000,E1 138.852} C_DIS
LIN {X 0.249,Y -541.881,Z 1519.571,A 0.000,B 0.000,C 90.000,E1 138.690} C_DIS
LIN {X -0.086,Y -543.041,Z 1519.570,A 0.000,B 0.000,C 90.000,E1 138.566} C_DIS
LIN {X 0.292,Y -544.587,Z 1519.568,A 0.000,B 0.000,C 90.000,E1 138.243} C_DIS
LIN {X -0.090,Y -545.796,Z 1519.567,A 0.000,B 0.000,C 90.000,E1 138.000} C_DIS
LIN {X 0.334,Y -547.627,Z 1519.563,A 0.000,B 0.000,C 90.000,E1 137.391} C_DIS
LIN {X -0.007,Y -548.992,Z 1519.560,A 0.000,B 0.000,C 90.000,E1 136.863} C_DIS
LIN {X 0.038,Y -550.077,Z 1519.557,A 0.000,B 0.000,C 90.000,E1 136.296} C_DIS
LIN {X -0.267,Y -551.287,Z 1519.553,A 0.000,B 0.000,C 90.000,E1 135.486} C_DIS
LIN {X 0.296,Y -552.831,Z 1519.545,A 0.000,B 0.000,C 90.000,E1 134.028} C_DIS
LIN {X 0.070,Y -553.909,Z 1519.539,A 0.000,B 0.000,C 90.000,E1 132.933} C_DIS
LIN {X -0.077,Y -555.106,Z 1519.531,A 0.000,B 0.000,C 90.000,E1 131.553} C_DIS
LIN {X -0.130,Y -556.367,Z 1519.522,A 0.000,B 0.000,C 90.000,E1 129.886} C_DIS
LIN {X 0.265,Y -557.437,Z 1519.512,A 0.000,B 0.000,C 90.000,E1 128.177} C_DIS
LIN {X 0.243,Y -558.258,Z 1519.505,A 0.000,B 0.000,C 90.000,E1 126.790} C_DIS
LIN {X -0.192,Y -558.796,Z 1519.498,A 0.000,B 0.000,C 90.000,E1 125.724} C_DIS
LIN {X -0.078,Y -559.286,Z 1519.491,A 0.000,B 0.000,C 90.000,E1 124.326} C_DIS
LIN {X -0.046,Y -559.484,Z 1519.484,A 0.000,B 0.000,C 90.000,E1 123.214} C_DIS
LIN {X -0.112,Y -559.574,Z 1519.472,A 0.000,B 0.000,C 90.000,E1 121.003} C_DIS
LIN {X 0.313,Y -560.015,Z 1519.460,A 0.000,B 0.000,C 90.000,E1 118.743} C_DIS
LIN {X -0.148,Y -560.372,Z 1519.451,A 0.000,B 0.000,C 90.000,E1 117.129} C_DIS
LIN {X 0.300,Y -560.641,Z 1519.445,A 0.000,B 0.000,C 90.000,E1 115.976} C_DIS
LIN {X -0.092,Y -560.965,Z 1519.434,A 0.000,B 0.000,C 90.000,E1 114.079} C_DIS
LIN {X 0.125,Y -561.198,Z 1519.428,A 0.000,B 0.000,C 90.000,E1 112.950} C_DIS
LIN {X 0.137,Y -561.553,Z 1519.415,A 0.000,B 0.000,C 90.000,E1 110.737} C_DIS
LIN {X -0.257,Y -561.805,Z 1519.408,A 0.000,B 0.000,C 90.000,E1 109.396} C_DIS
LIN {X 0.190,Y -562.104,Z 1519.398,A 0.000,B 0.000,C 90.000,E1 107.692} C_DIS
LIN {X -0.093,Y -562.486,Z 1519.388,A 0.000,B 0.000,C 90.000,E1 105.788} C_DIS
LIN {X -0.126,Y -562.810,Z 1519.380,A 0.000,B 0.000,C 90.000,E1 104.411} C_DIS
LIN {X -0.278,Y -563.238,Z 1519.371,A 0.000,B 0.000,C 90.000,E1 102.771} C_DIS
LIN {X -0.083,Y -564.022,Z 1519.359,A 0.000,B 0.000,C 90.000,E1 100.546} C_DIS
LIN {X -0.068,Y -564.938,Z 1519.346,A 0.000,B 0.000,C 90.000,E1 98.341} C_DIS
LIN {X 0.201,Y -565.602,Z 1519.337,A 0.000,B 0.000,C 90.000,E1 96.663} C_DIS
LIN {X 0.005,Y -566.465,Z 1519.327,A 0.000,B 0.000,C 90.000,E1 94.759} C_DIS
LIN {X 0.032,Y -567.066,Z 1519.319,A 0.000,B 0.000,C 90.000,E1 93.383} C_DIS
LIN {X 0.218,Y -567.878,Z 1519.310,A 0.000,B 0.000,C 90.000,E1 91.718} C_DIS
LIN {X -0.183,Y -568.717,Z 1519.301,A 0.000,B 0.000,C 90.000,E1 90.115} C_DIS
LIN {X 0.001,Y -569.550,Z 1519.292,A 0.000,B 0.000,C 90.000,E1 88.453} C_DIS
LIN {X 0.243,Y -570.428,Z 1519.282,A 0.000,B 0.000,C 90.000,E1 86.788} C_DIS
LIN {X 0.072,Y -571.459,Z 1519.272,A 0.000,B 0.000,C 90.000,E1 84.894} C_DIS
LIN {X -0.159,Y -572.415,Z 1519.263,A 0.000,B 0.000,C 90.000,E1 83.280} C_DIS
LIN {X 0.273,Y -573.507,Z 1519.254,A 0.000,B 0.000,C 90.000,E1 81.602} C_DIS
LIN {X 0.154,Y -574.625,Z 1519.245,A 0.000,B 0.000,C 90.000,E1 79.982} C_DIS
LIN {X 0.261,Y -575.837,Z 1519.235,A 0.000,B 0.000,C 90.000,E1 78.342} C_DIS
LIN {X 0.190,Y -576.882,Z 1519.228,A 0.000,B 0.000,C 90.000,E1 76.992} C_DIS
LIN {X 0.128,Y -577.929,Z 1519.220,A 0.000,B 0.000,C 90.000,E1 75.644} C_DIS
LIN {X 0.006,Y -578.680,Z 1519.214,A 0.000,B 0.000,C 90.000,E1 74.574} C_DIS
LIN {X 0.271,Y -579.539,Z 1519.207,A 0.000,B 0.000,C 90.000,E1 73.196} C_DIS
LIN {X 0.169,Y -580.259,Z 1519.201,A 0.000,B 0.000,C 90.000,E1 72.127} C_DIS
LIN {X 0.136,Y -581.473,Z 1519.190,A 0.000,B 0.000,C 90.000,E1 70.242} C_DIS
LIN {X 0.127,Y -582.512,Z 1519.180,A 0.000,B 0.000,C 90.000,E1 68.358} C_DIS
LIN {X 0.027,Y -583.571,Z 1519.169,A 0.000,B 0.000,C 90.000,E1 66.485} C_DIS
LIN {X 0.078,Y -584.733,Z 1519.157,A 0.000,B 0.000,C 90.000,E1 64.332} C_DIS
LIN {X -0.127,Y -585.763,Z 1519.149,A 0.000,B 0.000,C 90.000,E1 62.743} C_DIS
LIN {X 0.067,Y -586.769,Z 1519.141,A 0.000,B 0.000,C 90.000,E1 61.385} C_DIS
LIN {X -0.122,Y -587.582,Z 1519.135,A 0.000,B 0.000,C 90.000,E1 60.333} C_DIS
LIN {X -0.121,Y -588.505,Z 1519.128,A 0.000,B 0.000,C 90.000,E1 58.997} C_DIS
LIN {X -0.103,Y -589.411,Z 1519.120,A 0.000,B 0.000,C 90.000,E1 57.661} C_DIS
LIN {X 0.042,Y -590.147,Z 1519.114,A 0.000,B 0.000,C 90.000,E1 56.580} C_DIS
LIN {X -0.096,Y -591.121,Z 1519.107,A 0.000,B 0.000,C 90.000,E1 55.261} C_DIS
LIN {X 0.128,Y -591.833,Z 1519.100,A 0.000,B 0.000,C 90.000,E1 53.909} C_DIS
LIN {X -0.103,Y -592.441,Z 1519.092,A 0.000,B 0.000,C 90.000,E1 52.603} C_DIS
LIN {X -0.102,Y -593.102,Z 1519.083,A 0.000,B 0.000,C 90.000,E1 51.009} C_DIS
LIN {X 0.040,Y -593.868,Z 1519.073,A 0.000,B 0.000,C 90.000,E1 49.138} C_DIS
LIN {X -0.003,Y -594.174,Z 1519.067,A 0.000,B 0.000,C 90.000,E1 48.081} C_DIS
LIN {X 0.127,Y -594.135,Z 1519.060,A 0.000,B 0.000,C 90.000,E1 46.743} C_DIS
LIN {X -0.357,Y -593.987,Z 1519.054,A 0.000,B 0.000,C 90.000,E1 45.729} C_DIS
LIN {X -0.014,Y -593.592,Z 1519.048,A 0.000,B 0.000,C 90.000,E1 44.636} C_DIS
LIN {X -0.084,Y -592.957,Z 1519.042,A 0.000,B 0.000,C 90.000,E1 43.581} C_DIS
LIN {X 0.023,Y -591.786,Z 1519.035,A 0.000,B 0.000,C 90.000,E1 42.243} C_DIS
LIN {X 0.098,Y -590.364,Z 1519.027,A 0.000,B 0.000,C 90.000,E1 40.906} C_DIS
LIN {X 0.252,Y -589.398,Z 1519.023,A 0.000,B 0.000,C 90.000,E1 40.092} C_DIS
LIN {X 0.000,Y -589.005,Z 1519.021,A 0.000,B 0.000,C 90.000,E1 39.850} C_DIS
LIN {X -0.058,Y -587.859,Z 1519.018,A 0.000,B 0.000,C 90.000,E1 39.322} C_DIS
LIN {X 0.333,Y -586.416,Z 1519.016,A 0.000,B 0.000,C 90.000,E1 38.749} C_DIS
LIN {X -0.297,Y -585.446,Z 1519.014,A 0.000,B 0.000,C 90.000,E1 38.543} C_DIS
LIN {X -0.105,Y -584.222,Z 1519.013,A 0.000,B 0.000,C 90.000,E1 38.257} C_DIS
LIN {X 0.083,Y -582.672,Z 1519.011,A 0.000,B 0.000,C 90.000,E1 37.971} C_DIS
LIN {X -0.107,Y -581.682,Z 1519.010,A 0.000,B 0.000,C 90.000,E1 37.855} C_DIS
LIN {X -0.035,Y -579.936,Z 1519.009,A 0.000,B 0.000,C 90.000,E1 37.684} C_DIS
LIN {X -0.182,Y -578.886,Z 1519.009,A 0.000,B 0.000,C 90.000,E1 37.649} C_DIS
LIN {X 0.172,Y -578.360,Z 1519.009,A 0.000,B 0.000,C 90.000,E1 37.604} C_DIS
LIN {X 0.084,Y -403.933,Z 1519.009,A 0.000,B 0.000,C 90.000,E1 37.604} C_DIS
LIN {X 0.026,Y -395.851,Z 1518.985,A 0.000,B 0.000,C 90.000,E1 33.245} C_DIS
LIN {X -0.075,Y -393.797,Z 1518.977,A 0.000,B 0.000,C 90.000,E1 31.848} C_DIS
LIN {X -0.159,Y -386.381,Z 1518.953,A 0.000,B 0.000,C 90.000,E1 27.590} C_DIS
LIN {X -0.016,Y -382.674,Z 1518.937,A 0.000,B 0.000,C 90.000,E1 24.695} C_DIS
LIN {X -0.084,Y -376.020,Z 1518.911,A 0.000,B 0.000,C 90.000,E1 19.993} C_DIS
LIN {X 0.133,Y -373.552,Z 1518.897,A 0.000,B 0.000,C 90.000,E1 17.402} C_DIS
LIN {X -0.189,Y -367.975,Z 1518.868,A 0.000,B 0.000,C 90.000,E1 12.299} C_DIS
LIN {X 0.189,Y -366.550,Z 1518.856,A 0.000,B 0.000,C 90.000,E1 10.018} C_DIS
LIN {X -0.098,Y -365.840,Z 1518.852,A 0.000,B 0.000,C 90.000,E1 9.321} C_DIS
LIN {X -0.083,Y -361.397,Z 1518.817,A 0.000,B 0.000,C 90.000,E1 2.980} C_DIS
LIN {X 0.008,Y -360.907,Z 1518.802,A 0.000,B 0.000,C 90.000,E1 0.344} C_DIS
LIN {X 0.105,Y -360.314,Z 1518.795,A 0.000,B 0.000,C 90.000,E1 359.026} C_DIS
LIN {X -0.053,Y -359.426,Z 1518.770,A 0.000,B 0.000,C 90.000,E1 354.546} C_DIS
LIN {X 0.070,Y -358.890,Z 1518.759,A 0.000,B 0.000,C 90.000,E1 352.648} C_DIS
LIN {X -0.020,Y -359.563,Z 1518.726,A 0.000,B 0.000,C 90.000,E1 346.645} C_DIS
LIN {X 0.001,Y -361.801,Z 1518.684,A 0.000,B 0.000,C 90.000,E1 339.135} C_DIS
LIN {X -0.154,Y -362.053,Z 1518.680,A 0.000,B 0.000,C 90.000,E1 338.411} C_DIS
LIN {X 0.189,Y -365.980,Z 1518.643,A 0.000,B 0.000,C 90.000,E1 331.641} C_DIS
LIN {X 0.029,Y -366.387,Z 1518.639,A 0.000,B 0.000,C 90.000,E1 330.923} C_DIS
LIN {X -0.031,Y -371.355,Z 1518.604,A 0.000,B 0.000,C 90.000,E1 324.642} C_DIS
LIN {X -0.043,Y -371.766,Z 1518.602,A 0.000,B 0.000,C 90.000,E1 324.276} C_DIS
LIN {X 0.013,Y -377.358,Z 1518.567,A 0.000,B 0.000,C 90.000,E1 318.038} C_DIS
LIN {X 0.012,Y -378.235,Z 1518.563,A 0.000,B 0.000,C 90.000,E1 317.310} C_DIS
LIN {X 0.002,Y -383.940,Z 1518.531,A 0.000,B 0.000,C 90.000,E1 311.515} C_DIS
LIN {X 0.088,Y -384.893,Z 1518.527,A 0.000,B 0.000,C 90.000,E1 310.782} C_DIS
LIN {X 0.262,Y -390.610,Z 1518.495,A 0.000,B 0.000,C 90.000,E1 305.025} C_DIS
LIN {X 0.106,Y -391.104,Z 1518.493,A 0.000,B 0.000,C 90.000,E1 304.692} C_DIS
LIN {X 0.022,Y -391.648,Z 1518.489,A 0.000,B 0.000,C 90.000,E1 303.992} C_DIS
LIN {X -0.080,Y -396.825,Z 1518.459,A 0.000,B 0.000,C 90.000,E1 298.693} C_DIS
LIN {X -0.210,Y -397.120,Z 1518.457,A 0.000,B 0.000,C 90.000,E1 298.359} C_DIS
LIN {X -0.055,Y -401.597,Z 1518.426,A 0.000,B 0.000,C 90.000,E1 292.717} C_DIS
LIN {X 0.222,Y -404.659,Z 1518.395,A 0.000,B 0.000,C 90.000,E1 287.094} C_DIS
LIN {X -0.079,Y -404.735,Z 1518.391,A 0.000,B 0.000,C 90.000,E1 286.441} C_DIS
LIN {X 0.214,Y -406.099,Z 1518.364,A 0.000,B 0.000,C 90.000,E1 281.535} C_DIS
LIN {X -0.176,Y -406.094,Z 1518.362,A 0.000,B 0.000,C 90.000,E1 281.243} C_DIS
LIN {X -0.097,Y -405.680,Z 1518.333,A 0.000,B 0.000,C 90.000,E1 276.024} C_DIS
LIN {X -0.165,Y -405.058,Z 1518.328,A 0.000,B 0.000,C 90.000,E1 274.992} C_DIS
LIN {X -0.060,Y -403.497,Z 1518.304,A 0.000,B 0.000,C 90.000,E1 270.802} C_DIS
LIN {X -0.092,Y -403.288,Z 1518.302,A 0.000,B 0.000,C 90.000,E1 270.458} C_DIS
LIN {X 0.091,Y -398.931,Z 1518.271,A 0.000,B 0.000,C 90.000,E1 264.837} C_DIS
LIN {X -0.040,Y -393.108,Z 1518.242,A 0.000,B 0.000,C 90.000,E1 259.567} C_DIS
LIN {X -0.079,Y -392.835,Z 1518.240,A 0.000,B 0.000,C 90.000,E1 259.218} C_DIS
LIN {X 0.034,Y -385.993,Z 1518.212,A 0.000,B 0.000,C 90.000,E1 254.212} C_DIS
LIN {X -0.026,Y -385.267,Z 1518.208,A 0.000,B 0.000,C 90.000,E1 253.504} C_DIS
LIN {X -0.004,Y -384.768,Z 1518.206,A 0.000,B 0.000,C 90.000,E1 253.142} C_DIS
LIN {X 0.221,Y -377.973,Z 1518.182,A 0.000,B 0.000,C 90.000,E1 248.773} C_DIS
LIN {X -0.044,Y -376.233,Z 1518.174,A 0.000,B 0.000,C 90.000,E1 247.358} C_DIS
LIN {X 0.057,Y -374.944,Z 1518.170,A 0.000,B 0.000,C 90.000,E1 246.613} C_DIS
LIN {X -0.208,Y -368.417,Z 1518.148,A 0.000,B 0.000,C 90.000,E1 242.615} C_DIS
LIN {X 0.097,Y -366.047,Z 1518.137,A 0.000,B 0.000,C 90.000,E1 240.717} C_DIS
LIN {X 0.004,Y -359.196,Z 1518.115,A 0.000,B 0.000,C 90.000,E1 236.628} C_DIS
LIN {X 0.021,Y -355.842,Z 1518.100,A 0.000,B 0.000,C 90.000,E1 233.989} C_DIS
LIN {X -0.173,Y -348.793,Z 1518.075,A 0.000,B 0.000,C 90.000,E1 229.461} C_DIS
LIN {X -0.097,Y -346.185,Z 1518.062,A 0.000,B 0.000,C 90.000,E1 227.148} C_DIS
LIN {X -0.088,Y -345.065,Z 1518.058,A 0.000,B 0.000,C 90.000,E1 226.377} C_DIS
LIN {X 0.094,Y -338.586,Z 1518.030,A 0.000,B 0.000,C 90.000,E1 221.310} C_DIS
LIN {X 0.094,Y -336.840,Z 1518.019,A 0.000,B 0.000,C 90.000,E1 219.358} C_DIS
LIN {X 0.014,Y -330.861,Z 1517.988,A 0.000,B 0.000,C 90.000,E1 213.865} C_DIS
LIN {X 0.149,Y -329.296,Z 1517.975,A 0.000,B 0.000,C 90.000,E1 211.465} C_DIS
LIN {X -0.154,Y -324.669,Z 1517.942,A 0.000,B 0.000,C 90.000,E1 205.540} C_DIS
LIN {X 0.174,Y -323.837,Z 1517.928,A 0.000,B 0.000,C 90.000,E1 203.078} C_DIS
LIN {X -0.017,Y -321.124,Z 1517.881,A 0.000,B 0.000,C 90.000,E1 194.662} C_DIS
LIN {X 0.138,Y -320.932,Z 1517.877,A 0.000,B 0.000,C 90.000,E1 193.828} C_DIS
LIN {X -0.076,Y -321.562,Z 1517.832,A 0.000,B 0.000,C 90.000,E1 185.796} C_DIS
LIN {X -0.143,Y -324.415,Z 1517.790,A 0.000,B 0.000,C 90.000,E1 178.165} C_DIS
LIN {X -0.141,Y -325.376,Z 1517.783,A 0.000,B 0.000,C 90.000,E1 176.963} C_DIS
LIN {X -0.100,Y -329.112,Z 1517.750,A 0.000,B 0.000,C 90.000,E1 170.971} C_DIS
LIN {X 0.061,Y -334.260,Z 1517.726,A 0.000,B 0.000,C 90.000,E1 166.589} C_DIS
LIN {X 0.067,Y -335.488,Z 1517.719,A 0.000,B 0.000,C 90.000,E1 165.408} C_DIS
LIN {X 0.143,Y -340.932,Z 1517.695,A 0.000,B 0.000,C 90.000,E1 161.094} C_DIS
LIN {X -0.172,Y -342.138,Z 1517.691,A 0.000,B 0.000,C 90.000,E1 160.369} C_DIS
LIN {X -0.058,Y -347.939,Z 1517.667,A 0.000,B 0.000,C 90.000,E1 156.102} C_DIS
LIN {X -0.081,Y -354.259,Z 1517.648,A 0.000,B 0.000,C 90.000,E1 152.666} C_DIS
LIN {X -0.222,Y -361.406,Z 1517.625,A 0.000,B 0.000,C 90.000,E1 148.535} C_DIS
LIN {X 0.065,Y -368.758,Z 1517.606,A 0.000,B 0.000,C 90.000,E1 145.135} C_DIS
LIN {X 0.065,Y -377.029,Z 1517.584,A 0.000,B 0.000,C 90.000,E1 141.090} C_DIS
LIN {X 0.089,Y -380.392,Z 1517.576,A 0.000,B 0.000,C 90.000,E1 139.703} C_DIS
LIN {X 0.079,Y -538.285,Z 1517.576,A 0.000,B 0.000,C 90.000,E1 139.703} C_DIS
LIN {X 0.198,Y -539.878,Z 1517.576,A 0.000,B 0.000,C 90.000,E1 139.622} C_DIS
LIN {X -0.069,Y -541.350,Z 1517.575,A 0.000,B 0.000,C 90.000,E1 139.504} C_DIS
LIN {X 0.106,Y -543.092,Z 1517.574,A 0.000,B 0.000,C 90.000,E1 139.218} C_DIS
LIN {X 0.127,Y -544.473,Z 1517.572,A 0.000,B 0.000,C 90.000,E1 138.933} C_DIS
LIN {X -0.257,Y -545.543,Z 1517.570,A 0.000,B 0.000,C 90.000,E1 138.690} C_DIS
LIN {X 0.164,Y -547.304,Z 1517.567,A 0.000,B 0.000,C 90.000,E1 138.081} C_DIS
LIN {X -0.176,Y -548.626,Z 1517.564,A 0.000,B 0.000,C 90.000,E1 137.553} C_DIS
LIN {X -0.136,Y -549.660,Z 1517.561,A 0.000,B 0.000,C 90.000,E1 136.986} C_DIS
LIN {X -0.045,Y -550.819,Z 1517.556,A 0.000,B 0.000,C 90.000,E1 136.134} C_DIS
LIN {X -0.272,Y -552.479,Z 1517.549,A 0.000,B 0.000,C 90.000,E1 134.757} C_DIS
LIN {X -0.071,Y -553.895,Z 1517.541,A 0.000,B 0.000,C 90.000,E1 133.338} C_DIS
LIN {X 0.156,Y -555.115,Z 1517.533,A 0.000,B 0.000,C 90.000,E1 131.919} C_DIS
LIN {X -0.045,Y -555.957,Z 1517.527,A 0.000,B 0.000,C 90.000,E1 130.825} C_DIS
LIN {X -0.098,Y -556.928,Z 1517.519,A 0.000,B 0.000,C 90.000,E1 129.439} C_DIS
LIN {X 0.306,Y -557.958,Z 1517.510,A 0.000,B 0.000,C 90.000,E1 127.729} C_DIS
LIN {X -0.045,Y -558.770,Z 1517.502,A 0.000,B 0.000,C 90.000,E1 126.377} C_DIS
LIN {X 0.075,Y -559.256,Z 1517.494,A 0.000,B 0.000,C 90.000,E1 124.978} C_DIS
LIN {X 0.116,Y -559.566,Z 1517.488,A 0.000,B 0.000,C 90.000,E1 123.865} C_DIS
LIN {X 0.070,Y -559.614,Z 1517.484,A 0.000,B 0.000,C 90.000,E1 123.038} C_DIS
LIN {X 0.102,Y -559.721,Z 1517.470,A 0.000,B 0.000,C 90.000,E1 120.541} C_DIS
LIN {X 0.180,Y -560.073,Z 1517.461,A 0.000,B 0.000,C 90.000,E1 118.871} C_DIS
LIN {X -0.080,Y -560.381,Z 1517.453,A 0.000,B 0.000,C 90.000,E1 117.513} C_DIS
LIN {X -0.034,Y -560.749,Z 1517.444,A 0.000,B 0.000,C 90.000,E1 115.848} C_DIS
LIN {X 0.089,Y -561.098,Z 1517.433,A 0.000,B 0.000,C 90.000,E1 113.898} C_DIS
LIN {X 0.105,Y -561.346,Z 1517.425,A 0.000,B 0.000,C 90.000,E1 112.514} C_DIS
LIN {X 0.014,Y -561.645,Z 1517.416,A 0.000,B 0.000,C 90.000,E1 110.865} C_DIS
LIN {X -0.188,Y -561.893,Z 1517.408,A 0.000,B 0.000,C 90.000,E1 109.504} C_DIS
LIN {X -0.231,Y -562.141,Z 1517.401,A 0.000,B 0.000,C 90.000,E1 108.127} C_DIS
LIN {X -0.041,Y -562.582,Z 1517.388,A 0.000,B 0.000,C 90.000,E1 105.898} C_DIS
LIN {X -0.221,Y -562.911,Z 1517.381,A 0.000,B 0.000,C 90.000,E1 104.537} C_DIS
LIN {X -0.078,Y -563.412,Z 1517.370,A 0.000,B 0.000,C 90.000,E1 102.591} C_DIS
LIN {X -0.048,Y -564.102,Z 1517.359,A 0.000,B 0.000,C 90.000,E1 100.658} C_DIS
LIN {X -0.202,Y -564.934,Z 1517.349,A 0.000,B 0.000,C 90.000,E1 98.746} C_DIS
LIN {X 0.067,Y -565.579,Z 1517.339,A 0.000,B 0.000,C 90.000,E1 97.068} C_DIS
LIN {X -0.225,Y -566.313,Z 1517.330,A 0.000,B 0.000,C 90.000,E1 95.448} C_DIS
LIN {X -0.205,Y -566.995,Z 1517.323,A 0.000,B 0.000,C 90.000,E1 94.073} C_DIS
LIN {X 0.231,Y -568.049,Z 1517.310,A 0.000,B 0.000,C 90.000,E1 91.835} C_DIS
LIN {X -0.151,Y -568.927,Z 1517.301,A 0.000,B 0.000,C 90.000,E1 90.229} C_DIS
LIN {X 0.166,Y -569.920,Z 1517.291,A 0.000,B 0.000,C 90.000,E1 88.282} C_DIS
LIN {X -0.027,Y -570.921,Z 1517.280,A 0.000,B 0.000,C 90.000,E1 86.388} C_DIS
LIN {X 0.248,Y -571.850,Z 1517.271,A 0.000,B 0.000,C 90.000,E1 84.723} C_DIS
LIN {X 0.210,Y -573.001,Z 1517.260,A 0.000,B 0.000,C 90.000,E1 82.818} C_DIS
LIN {X 0.197,Y -574.325,Z 1517.250,A 0.000,B 0.000,C 90.000,E1 80.914} C_DIS
LIN {X -0.179,Y -575.687,Z 1517.239,A 0.000,B 0.000,C 90.000,E1 79.050} C_DIS
LIN {X -0.050,Y -576.945,Z 1517.230,A 0.000,B 0.000,C 90.000,E1 77.409} C_DIS
LIN {X 0.241,Y -578.169,Z 1517.221,A 0.000,B 0.000,C 90.000,E1 75.755} C_DIS
LIN {X -0.216,Y -579.093,Z 1517.214,A 0.000,B 0.000,C 90.000,E1 74.448} C_DIS
LIN {X 0.239,Y -579.798,Z 1517.208,A 0.000,B 0.000,C 90.000,E1 73.323} C_DIS
LIN {X -0.032,Y -580.687,Z 1517.200,A 0.000,B 0.000,C 90.000,E1 72.000} C_DIS
LIN {X -0.049,Y -581.856,Z 1517.190,A 0.000,B 0.000,C 90.000,E1 70.115} C_DIS
LIN {X -0.046,Y -582.898,Z 1517.179,A 0.000,B 0.000,C 90.000,E1 68.230} C_DIS
LIN {X -0.132,Y -583.975,Z 1517.169,A 0.000,B 0.000,C 90.000,E1 66.357} C_DIS
LIN {X 0.215,Y -585.509,Z 1517.154,A 0.000,B 0.000,C 90.000,E1 63.640} C_DIS
LIN {X 0.053,Y -587.028,Z 1517.142,A 0.000,B 0.000,C 90.000,E1 61.513} C_DIS
LIN {X -0.250,Y -588.033,Z 1517.134,A 0.000,B 0.000,C 90.000,E1 60.205} C_DIS
LIN {X -0.243,Y -588.942,Z 1517.127,A 0.000,B 0.000,C 90.000,E1 58.869} C_DIS
LIN {X 0.174,Y -590.244,Z 1517.117,A 0.000,B 0.000,C 90.000,E1 56.962} C_DIS
LIN {X 0.131,Y -591.571,Z 1517.106,A 0.000,B 0.000,C 90.000,E1 55.102} C_DIS
LIN {X 0.021,Y -592.268,Z 1517.099,A 0.000,B 0.000,C 90.000,E1 53.783} C_DIS
LIN {X -0.208,Y -592.844,Z 1517.091,A 0.000,B 0.000,C 90.000,E1 52.477} C_DIS
LIN {X -0.208,Y -593.570,Z 1517.083,A 0.000,B 0.000,C 90.000,E1 50.884} C_DIS
LIN {X -0.299,Y -594.417,Z 1517.071,A 0.000,B 0.000,C 90.000,E1 48.771} C_DIS
LIN {X -0.107,Y -594.620,Z 1517.066,A 0.000,B 0.000,C 90.000,E1 47.957} C_DIS
LIN {X 0.021,Y -594.530,Z 1517.059,A 0.000,B 0.000,C 90.000,E1 46.620} C_DIS
LIN {X -0.049,Y -594.359,Z 1517.053,A 0.000,B 0.000,C 90.000,E1 45.567} C_DIS
LIN {X -0.347,Y -593.817,Z 1517.046,A 0.000,B 0.000,C 90.000,E1 44.271} C_DIS
LIN {X 0.034,Y -593.530,Z 1517.043,A 0.000,B 0.000,C 90.000,E1 43.704} C_DIS
LIN {X -0.095,Y -592.069,Z 1517.034,A 0.000,B 0.000,C 90.000,E1 42.123} C_DIS
LIN {X 0.034,Y -590.711,Z 1517.027,A 0.000,B 0.000,C 90.000,E1 40.782} C_DIS
LIN {X -0.053,Y -589.402,Z 1517.021,A 0.000,B 0.000,C 90.000,E1 39.725} C_DIS
LIN {X 0.095,Y -588.079,Z 1517.016,A 0.000,B 0.000,C 90.000,E1 38.910} C_DIS
LIN {X -0.165,Y -587.469,Z 1517.015,A 0.000,B 0.000,C 90.000,E1 38.669} C_DIS
LIN {X 0.032,Y -586.721,Z 1517.013,A 0.000,B 0.000,C 90.000,E1 38.382} C_DIS
LIN {X -0.043,Y -584.828,Z 1517.010,A 0.000,B 0.000,C 90.000,E1 37.855} C_DIS
LIN {X -0.212,Y -583.645,Z 1517.009,A 0.000,B 0.000,C 90.000,E1 37.604} C_DIS
LIN {X -0.025,Y -582.134,Z 1517.007,A 0.000,B 0.000,C 90.000,E1 37.317} C_DIS
LIN {X 0.241,Y -581.206,Z 1517.007,A 0.000,B 0.000,C 90.000,E1 37.156} C_DIS
LIN {X -0.156,Y -579.661,Z 1517.006,A 0.000,B 0.000,C 90.000,E1 37.030} C_DIS
LIN {X -0.079,Y -578.612,Z 1517.005,A 0.000,B 0.000,C 90.000,E1 36.950} C_DIS
LIN {X 0.294,Y -577.364,Z 1517.005,A 0.000,B 0.000,C 90.000,E1 36.870} C_DIS
LIN {X 0.179,Y -402.413,Z 1517.005,A 0.000,B 0.000,C 90.000,E1 36.870} C_DIS
LIN {X 0.003,Y -394.319,Z 1516.979,A 0.000,B 0.000,C 90.000,E1 32.212} C_DIS
LIN {X -0.130,Y -393.829,Z 1516.977,A 0.000,B 0.000,C 90.000,E1 31.878} C_DIS
LIN {X -0.008,Y -386.414,Z 1516.953,A 0.000,B 0.000,C 90.000,E1 27.590} C_DIS
LIN {X -0.025,Y -382.713,Z 1516.937,A 0.000,B 0.000,C 90.000,E1 24.719} C_DIS
LIN {X 0.066,Y -376.046,Z 1516.911,A 0.000,B 0.000,C 90.000,E1 19.993} C_DIS
LIN {X -0.074,Y -373.580,Z 1516.897,A 0.000,B 0.000,C 90.000,E1 17.457} C_DIS
LIN {X -0.040,Y -367.993,Z 1516.868,A 0.000,B 0.000,C 90.000,E1 12.299} C_DIS
LIN {X -0.022,Y -366.561,Z 1516.856,A 0.000,B 0.000,C 90.000,E1 10.074} C_DIS
LIN {X 0.050,Y -365.865,Z 1516.852,A 0.000,B 0.000,C 90.000,E1 9.321} C_DIS
LIN {X 0.065,Y -361.405,Z 1516.817,A 0.000,B 0.000,C 90.000,E1 2.980} C_DIS
LIN {X 0.155,Y -360.907,Z 1516.802,A 0.000,B 0.000,C 90.000,E1 0.344} C_DIS
LIN {X -0.058,Y -360.492,Z 1516.797,A 0.000,B 0.000,C 90.000,E1 359.427} C_DIS
LIN {X -0.053,Y -359.426,Z 1516.770,A 0.000,B 0.000,C 90.000,E1 354.546} C_DIS
LIN {X 0.070,Y -358.890,Z 1516.759,A 0.000,B 0.000,C 90.000,E1 352.648} C_DIS
LIN {X -0.020,Y -359.563,Z 1516.726,A 0.000,B 0.000,C 90.000,E1 346.645} C_DIS
LIN {X 0.001,Y -361.801,Z 1516.684,A 0.000,B 0.000,C 90.000,E1 339.135} C_DIS
LIN {X -0.154,Y -362.053,Z 1516.680,A 0.000,B 0.000,C 90.000,E1 338.411} C_DIS
LIN {X 0.189,Y -365.980,Z 1516.643,A 0.000,B 0.000,C 90.000,E1 331.641} C_DIS
LIN {X 0.029,Y -366.387,Z 1516.639,A 0.000,B 0.000,C 90.000,E1 330.923} C_DIS
LIN {X -0.031,Y -371.355,Z 1516.604,A 0.000,B 0.000,C 90.000,E1 324.642} C_DIS
LIN {X -0.043,Y -371.766,Z 1516.602,A 0.000,B 0.000,C 90.000,E1 324.276} C_DIS
LIN {X 0.013,Y -377.358,Z 1516.567,A 0.000,B 0.000,C 90.000,E1 318.038} C_DIS
LIN {X 0.012,Y -378.235,Z 1516.563,A 0.000,B 0.000,C 90.000,E1 317.310} C_DIS
LIN {X 0.002,Y -383.940,Z 1516.531,A 0.000,B 0.000,C 90.000,E1 311.515} C_DIS
LIN {X 0.088,Y -384.893,Z 1516.527,A 0.000,B 0.000,C 90.000,E1 310.782} C_DIS
LIN {X 0.262,Y -390.610,Z 1516.495,A 0.000,B 0.000,C 90.000,E1 305.025} C_DIS
LIN {X 0.106,Y -391.104,Z 1516.493,A 0.000,B 0.000,C 90.000,E1 304.692} C_DIS
LIN {X 0.022,Y -391.648,Z 1516.489,A 0.000,B 0.000,C 90.000,E1 303.992} C_DIS
LIN {X -0.080,Y -396.825,Z 1516.459,A 0.000,B 0.000,C 90.000,E1 298.693} C_DIS
LIN {X -0.210,Y -397.120,Z 1516.457,A 0.000,B 0.000,C 90.000,E1 298.359} C_DIS
LIN {X -0.055,Y -401.597,Z 1516.426,A 0.000,B 0.000,C 90.000,E1 292.717} C_DIS
LIN {X 0.222,Y -404.659,Z 1516.395,A 0.000,B 0.000,C 90.000,E1 287.094} C_DIS
LIN {X -0.079,Y -404.735,Z 1516.391,A 0.000,B 0.000,C 90.000,E1 286.441} C_DIS
LIN {X 0.214,Y -406.099,Z 1516.364,A 0.000,B 0.000,C 90.000,E1 281.535} C_DIS
LIN {X -0.176,Y -406.094,Z 1516.362,A 0.000,B 0.000,C 90.000,E1 281.243} C_DIS
LIN {X -0.097,Y -405.680,Z 1516.333,A 0.000,B 0.000,C 90.000,E1 276.024} C_DIS
LIN {X -0.165,Y -405.058,Z 1516.328,A 0.000,B 0.000,C 90.000,E1 274.992} C_DIS
LIN {X -0.060,Y -403.497,Z 1516.304,A 0.000,B 0.000,C 90.000,E1 270.802} C_DIS
LIN {X -0.092,Y -403.288,Z 1516.302,A 0.000,B 0.000,C 90.000,E1 270.458} C_DIS
LIN {X 0.091,Y -398.931,Z 1516.271,A 0.000,B 0.000,C 90.000,E1 264.837} C_DIS
LIN {X -0.040,Y -393.108,Z 1516.242,A 0.000,B 0.000,C 90.000,E1 259.567} C_DIS
LIN {X -0.079,Y -392.835,Z 1516.240,A 0.000,B 0.000,C 90.000,E1 259.218} C_DIS
LIN {X 0.034,Y -385.993,Z 1516.212,A 0.000,B 0.000,C 90.000,E1 254.212} C_DIS
LIN {X -0.026,Y -385.267,Z 1516.208,A 0.000,B 0.000,C 90.000,E1 253.504} C_DIS
LIN {X -0.004,Y -384.768,Z 1516.206,A 0.000,B 0.000,C 90.000,E1 253.142} C_DIS
LIN {X 0.221,Y -377.973,Z 1516.182,A 0.000,B 0.000,C 90.000,E1 248.773} C_DIS
LIN {X -0.044,Y -376.233,Z 1516.174,A 0.000,B 0.000,C 90.000,E1 247.358} C_DIS
LIN {X 0.057,Y -374.944,Z 1516.170,A 0.000,B 0.000,C 90.000,E1 246.613} C_DIS
LIN {X -0.208,Y -368.417,Z 1516.148,A 0.000,B 0.000,C 90.000,E1 242.615} C_DIS
LIN {X 0.097,Y -366.047,Z 1516.137,A 0.000,B 0.000,C 90.000,E1 240.717} C_DIS
LIN {X 0.004,Y -359.196,Z 1516.115,A 0.000,B 0.000,C 90.000,E1 236.628} C_DIS
LIN {X 0.021,Y -355.842,Z 1516.100,A 0.000,B 0.000,C 90.000,E1 233.989} C_DIS
LIN {X -0.173,Y -348.793,Z 1516.075,A 0.000,B 0.000,C 90.000,E1 229.461} C_DIS
LIN {X -0.097,Y -346.185,Z 1516.062,A 0.000,B 0.000,C 90.000,E1 227.148} C_DIS
LIN {X -0.088,Y -345.065,Z 1516.058,A 0.000,B 0.000,C 90.000,E1 226.377} C_DIS
LIN {X 0.094,Y -338.586,Z 1516.030,A 0.000,B 0.000,C 90.000,E1 221.310} C_DIS
LIN {X 0.094,Y -336.840,Z 1516.019,A 0.000,B 0.000,C 90.000,E1 219.358} C_DIS
LIN {X 0.014,Y -330.861,Z 1515.988,A 0.000,B 0.000,C 90.000,E1 213.865} C_DIS
LIN {X 0.149,Y -329.296,Z 1515.975,A 0.000,B 0.000,C 90.000,E1 211.465} C_DIS
LIN {X -0.154,Y -324.669,Z 1515.942,A 0.000,B 0.000,C 90.000,E1 205.540} C_DIS
LIN {X 0.174,Y -323.837,Z 1515.928,A 0.000,B 0.000,C 90.000,E1 203.078} C_DIS
LIN {X -0.017,Y -321.124,Z 1515.881,A 0.000,B 0.000,C 90.000,E1 194.662} C_DIS
LIN {X 0.138,Y -320.932,Z 1515.877,A 0.000,B 0.000,C 90.000,E1 193.828} C_DIS
LIN {X -0.076,Y -321.562,Z 1515.832,A 0.000,B 0.000,C 90.000,E1 185.796} C_DIS
LIN {X -0.143,Y -324.415,Z 1515.790,A 0.000,B 0.000,C 90.000,E1 178.165} C_DIS
LIN {X -0.141,Y -325.376,Z 1515.783,A 0.000,B 0.000,C 90.000,E1 176.963} C_DIS
LIN {X -0.100,Y -329.112,Z 1515.750,A 0.000,B 0.000,C 90.000,E1 170.971} C_DIS
LIN {X 0.061,Y -334.260,Z 1515.726,A 0.000,B 0.000,C 90.000,E1 166.589} C_DIS
LIN {X 0.067,Y -335.488,Z 1515.719,A 0.000,B 0.000,C 90.000,E1 165.408} C_DIS
LIN {X 0.143,Y -340.932,Z 1515.695,A 0.000,B 0.000,C 90.000,E1 161.094} C_DIS
LIN {X -0.172,Y -342.138,Z 1515.691,A 0.000,B 0.000,C 90.000,E1 160.369} C_DIS
LIN {X -0.058,Y -347.939,Z 1515.667,A 0.000,B 0.000,C 90.000,E1 156.102} C_DIS
LIN {X -0.081,Y -354.259,Z 1515.648,A 0.000,B 0.000,C 90.000,E1 152.666} C_DIS
LIN {X -0.222,Y -361.406,Z 1515.625,A 0.000,B 0.000,C 90.000,E1 148.535} C_DIS
LIN {X 0.065,Y -368.758,Z 1515.606,A 0.000,B 0.000,C 90.000,E1 145.135} C_DIS
LIN {X 0.065,Y -377.029,Z 1515.584,A 0.000,B 0.000,C 90.000,E1 141.090} C_DIS
LIN {X 0.064,Y -378.387,Z 1515.581,A 0.000,B 0.000,C 90.000,E1 140.517} C_DIS
LIN {X 0.044,Y -537.362,Z 1515.581,A 0.000,B 0.000,C 90.000,E1 140.517} C_DIS
LIN {X 0.137,Y -539.935,Z 1515.580,A 0.000,B 0.000,C 90.000,E1 140.356} C_DIS
LIN {X -0.133,Y -541.378,Z 1515.579,A 0.000,B 0.000,C 90.000,E1 140.194} C_DIS
LIN {X -0.117,Y -542.947,Z 1515.577,A 0.000,B 0.000,C 90.000,E1 139.908} C_DIS
LIN {X -0.095,Y -544.180,Z 1515.576,A 0.000,B 0.000,C 90.000,E1 139.622} C_DIS
LIN {X -0.098,Y -546.116,Z 1515.573,A 0.000,B 0.000,C 90.000,E1 139.057} C_DIS
LIN {X -0.032,Y -547.559,Z 1515.569,A 0.000,B 0.000,C 90.000,E1 138.485} C_DIS
LIN {X -0.004,Y -548.729,Z 1515.566,A 0.000,B 0.000,C 90.000,E1 137.919} C_DIS
LIN {X 0.079,Y -549.985,Z 1515.562,A 0.000,B 0.000,C 90.000,E1 137.067} C_DIS
LIN {X 0.236,Y -551.740,Z 1515.554,A 0.000,B 0.000,C 90.000,E1 135.648} C_DIS
LIN {X -0.015,Y -553.002,Z 1515.548,A 0.000,B 0.000,C 90.000,E1 134.555} C_DIS
LIN {X -0.193,Y -554.413,Z 1515.540,A 0.000,B 0.000,C 90.000,E1 133.176} C_DIS
LIN {X -0.023,Y -555.347,Z 1515.534,A 0.000,B 0.000,C 90.000,E1 132.043} C_DIS
LIN {X 0.194,Y -556.175,Z 1515.527,A 0.000,B 0.000,C 90.000,E1 130.906} C_DIS
LIN {X -0.284,Y -557.125,Z 1515.520,A 0.000,B 0.000,C 90.000,E1 129.564} C_DIS
LIN {X -0.226,Y -558.158,Z 1515.510,A 0.000,B 0.000,C 90.000,E1 127.890} C_DIS
LIN {X -0.149,Y -559.074,Z 1515.501,A 0.000,B 0.000,C 90.000,E1 126.217} C_DIS
LIN {X -0.030,Y -559.536,Z 1515.493,A 0.000,B 0.000,C 90.000,E1 124.818} C_DIS
LIN {X 0.009,Y -559.756,Z 1515.487,A 0.000,B 0.000,C 90.000,E1 123.706} C_DIS
LIN {X -0.040,Y -559.746,Z 1515.483,A 0.000,B 0.000,C 90.000,E1 122.880} C_DIS
LIN {X -0.229,Y -559.901,Z 1515.467,A 0.000,B 0.000,C 90.000,E1 120.129} C_DIS
LIN {X -0.017,Y -560.134,Z 1515.461,A 0.000,B 0.000,C 90.000,E1 118.999} C_DIS
LIN {X 0.220,Y -560.437,Z 1515.453,A 0.000,B 0.000,C 90.000,E1 117.590} C_DIS
LIN {X 0.075,Y -560.852,Z 1515.443,A 0.000,B 0.000,C 90.000,E1 115.668} C_DIS
LIN {X -0.104,Y -561.174,Z 1515.433,A 0.000,B 0.000,C 90.000,E1 114.027} C_DIS
LIN {X 0.119,Y -561.378,Z 1515.427,A 0.000,B 0.000,C 90.000,E1 112.898} C_DIS
LIN {X 0.145,Y -561.768,Z 1515.415,A 0.000,B 0.000,C 90.000,E1 110.684} C_DIS
LIN {X -0.055,Y -562.030,Z 1515.407,A 0.000,B 0.000,C 90.000,E1 109.322} C_DIS
LIN {X -0.232,Y -562.222,Z 1515.401,A 0.000,B 0.000,C 90.000,E1 108.236} C_DIS
LIN {X 0.186,Y -562.583,Z 1515.391,A 0.000,B 0.000,C 90.000,E1 106.260} C_DIS
LIN {X 0.011,Y -562.942,Z 1515.383,A 0.000,B 0.000,C 90.000,E1 104.898} C_DIS
LIN {X 0.164,Y -563.424,Z 1515.372,A 0.000,B 0.000,C 90.000,E1 102.952} C_DIS
LIN {X 0.209,Y -564.098,Z 1515.361,A 0.000,B 0.000,C 90.000,E1 101.018} C_DIS
LIN {X -0.234,Y -565.052,Z 1515.349,A 0.000,B 0.000,C 90.000,E1 98.859} C_DIS
LIN {X 0.195,Y -565.797,Z 1515.339,A 0.000,B 0.000,C 90.000,E1 96.891} C_DIS
LIN {X -0.052,Y -566.751,Z 1515.328,A 0.000,B 0.000,C 90.000,E1 94.992} C_DIS
LIN {X 0.024,Y -567.376,Z 1515.320,A 0.000,B 0.000,C 90.000,E1 93.612} C_DIS
LIN {X -0.111,Y -568.517,Z 1515.308,A 0.000,B 0.000,C 90.000,E1 91.432} C_DIS
LIN {X 0.072,Y -569.394,Z 1515.299,A 0.000,B 0.000,C 90.000,E1 89.771} C_DIS
LIN {X -0.153,Y -570.423,Z 1515.288,A 0.000,B 0.000,C 90.000,E1 87.879} C_DIS
LIN {X 0.209,Y -571.439,Z 1515.278,A 0.000,B 0.000,C 90.000,E1 85.931} C_DIS
LIN {X -0.209,Y -572.245,Z 1515.270,A 0.000,B 0.000,C 90.000,E1 84.609} C_DIS
LIN {X -0.241,Y -573.420,Z 1515.259,A 0.000,B 0.000,C 90.000,E1 82.704} C_DIS
LIN {X -0.160,Y -574.761,Z 1515.249,A 0.000,B 0.000,C 90.000,E1 80.792} C_DIS
LIN {X 0.263,Y -576.344,Z 1515.237,A 0.000,B 0.000,C 90.000,E1 78.578} C_DIS
LIN {X -0.151,Y -577.595,Z 1515.228,A 0.000,B 0.000,C 90.000,E1 76.992} C_DIS
LIN {X -0.201,Y -578.601,Z 1515.220,A 0.000,B 0.000,C 90.000,E1 75.644} C_DIS
LIN {X -0.100,Y -579.530,Z 1515.213,A 0.000,B 0.000,C 90.000,E1 74.283} C_DIS
LIN {X -0.037,Y -580.221,Z 1515.207,A 0.000,B 0.000,C 90.000,E1 73.196} C_DIS
LIN {X 0.257,Y -581.112,Z 1515.199,A 0.000,B 0.000,C 90.000,E1 71.819} C_DIS
LIN {X 0.250,Y -582.251,Z 1515.189,A 0.000,B 0.000,C 90.000,E1 69.934} C_DIS
LIN {X -0.281,Y -583.287,Z 1515.178,A 0.000,B 0.000,C 90.000,E1 68.103} C_DIS
LIN {X -0.228,Y -584.214,Z 1515.169,A 0.000,B 0.000,C 90.000,E1 66.485} C_DIS
LIN {X -0.038,Y -585.197,Z 1515.159,A 0.000,B 0.000,C 90.000,E1 64.588} C_DIS
LIN {X -0.114,Y -586.105,Z 1515.151,A 0.000,B 0.000,C 90.000,E1 63.256} C_DIS
LIN {X -0.146,Y -587.459,Z 1515.141,A 0.000,B 0.000,C 90.000,E1 61.385} C_DIS
LIN {X -0.326,Y -588.292,Z 1515.135,A 0.000,B 0.000,C 90.000,E1 60.333} C_DIS
LIN {X 0.380,Y -589.354,Z 1515.126,A 0.000,B 0.000,C 90.000,E1 58.663} C_DIS
LIN {X -0.207,Y -590.491,Z 1515.117,A 0.000,B 0.000,C 90.000,E1 57.120} C_DIS
LIN {X -0.254,Y -591.849,Z 1515.107,A 0.000,B 0.000,C 90.000,E1 55.261} C_DIS
LIN {X -0.017,Y -592.586,Z 1515.099,A 0.000,B 0.000,C 90.000,E1 53.909} C_DIS
LIN {X 0.235,Y -593.151,Z 1515.092,A 0.000,B 0.000,C 90.000,E1 52.557} C_DIS
LIN {X -0.222,Y -593.886,Z 1515.083,A 0.000,B 0.000,C 90.000,E1 51.009} C_DIS
LIN {X 0.155,Y -594.794,Z 1515.072,A 0.000,B 0.000,C 90.000,E1 48.852} C_DIS
LIN {X 0.120,Y -594.976,Z 1515.066,A 0.000,B 0.000,C 90.000,E1 47.796} C_DIS
LIN {X 0.051,Y -594.932,Z 1515.060,A 0.000,B 0.000,C 90.000,E1 46.743} C_DIS
LIN {X 0.003,Y -594.771,Z 1515.054,A 0.000,B 0.000,C 90.000,E1 45.688} C_DIS
LIN {X -0.068,Y -594.418,Z 1515.048,A 0.000,B 0.000,C 90.000,E1 44.636} C_DIS
LIN {X 0.283,Y -593.818,Z 1515.042,A 0.000,B 0.000,C 90.000,E1 43.542} C_DIS
LIN {X -0.239,Y -592.353,Z 1515.033,A 0.000,B 0.000,C 90.000,E1 42.000} C_DIS
LIN {X 0.085,Y -591.274,Z 1515.027,A 0.000,B 0.000,C 90.000,E1 40.906} C_DIS
LIN {X 0.000,Y -590.015,Z 1515.021,A 0.000,B 0.000,C 90.000,E1 39.850} C_DIS
LIN {X 0.351,Y -588.541,Z 1515.016,A 0.000,B 0.000,C 90.000,E1 38.749} C_DIS
LIN {X -0.077,Y -587.424,Z 1515.013,A 0.000,B 0.000,C 90.000,E1 38.257} C_DIS
LIN {X -0.145,Y -585.992,Z 1515.010,A 0.000,B 0.000,C 90.000,E1 37.729} C_DIS
LIN {X 0.238,Y -584.059,Z 1515.007,A 0.000,B 0.000,C 90.000,E1 37.156} C_DIS
LIN {X -0.127,Y -582.065,Z 1515.004,A 0.000,B 0.000,C 90.000,E1 36.790} C_DIS
LIN {X 0.051,Y -580.347,Z 1515.003,A 0.000,B 0.000,C 90.000,E1 36.503} C_DIS
LIN {X 0.192,Y -578.663,Z 1515.002,A 0.000,B 0.000,C 90.000,E1 36.297} C_DIS
LIN {X 0.027,Y -577.261,Z 1515.001,A 0.000,B 0.000,C 90.000,E1 36.217} C_DIS
LIN {X 0.151,Y -576.209,Z 1515.001,A 0.000,B 0.000,C 90.000,E1 36.171} C_DIS
LIN {X 0.082,Y -400.981,Z 1515.001,A 0.000,B 0.000,C 90.000,E1 36.171} C_DIS
LIN {X 0.048,Y -393.866,Z 1514.977,A 0.000,B 0.000,C 90.000,E1 31.878} C_DIS
LIN {X -0.174,Y -386.452,Z 1514.953,A 0.000,B 0.000,C 90.000,E1 27.641} C_DIS
LIN {X -0.197,Y -382.758,Z 1514.938,A 0.000,B 0.000,C 90.000,E1 24.771} C_DIS
LIN {X -0.112,Y -376.076,Z 1514.911,A 0.000,B 0.000,C 90.000,E1 20.047} C_DIS
LIN {X 0.101,Y -373.610,Z 1514.897,A 0.000,B 0.000,C 90.000,E1 17.457} C_DIS
LIN {X 0.134,Y -368.014,Z 1514.869,A 0.000,B 0.000,C 90.000,E1 12.299} C_DIS
LIN {X 0.151,Y -366.575,Z 1514.856,A 0.000,B 0.000,C 90.000,E1 10.074} C_DIS
LIN {X 0.007,Y -366.303,Z 1514.854,A 0.000,B 0.000,C 90.000,E1 9.726} C_DIS
LIN {X -0.114,Y -361.702,Z 1514.821,A 0.000,B 0.000,C 90.000,E1 3.784} C_DIS
LIN {X -0.033,Y -360.909,Z 1514.802,A 0.000,B 0.000,C 90.000,E1 0.401} C_DIS
LIN {X 0.137,Y -360.684,Z 1514.799,A 0.000,B 0.000,C 90.000,E1 359.771} C_DIS
LIN {X -0.053,Y -359.426,Z 1514.770,A 0.000,B 0.000,C 90.000,E1 354.546} C_DIS
LIN {X 0.070,Y -358.890,Z 1514.759,A 0.000,B 0.000,C 90.000,E1 352.648} C_DIS
LIN {X -0.020,Y -359.563,Z 1514.726,A 0.000,B 0.000,C 90.000,E1 346.645} C_DIS
LIN {X 0.001,Y -361.801,Z 1514.684,A 0.000,B 0.000,C 90.000,E1 339.135} C_DIS
LIN {X -0.154,Y -362.053,Z 1514.680,A 0.000,B 0.000,C 90.000,E1 338.411} C_DIS
LIN {X 0.189,Y -365.980,Z 1514.643,A 0.000,B 0.000,C 90.000,E1 331.641} C_DIS
LIN {X 0.029,Y -366.387,Z 1514.639,A 0.000,B 0.000,C 90.000,E1 330.923} C_DIS
LIN {X -0.031,Y -371.355,Z 1514.604,A 0.000,B 0.000,C 90.000,E1 324.642} C_DIS
LIN {X -0.043,Y -371.766,Z 1514.602,A 0.000,B 0.000,C 90.000,E1 324.276} C_DIS
LIN {X 0.013,Y -377.358,Z 1514.567,A 0.000,B 0.000,C 90.000,E1 318.038} C_DIS
LIN {X 0.012,Y -378.235,Z 1514.563,A 0.000,B 0.000,C 90.000,E1 317.310} C_DIS
LIN {X 0.002,Y -383.940,Z 1514.531,A 0.000,B 0.000,C 90.000,E1 311.515} C_DIS
LIN {X 0.088,Y -384.893,Z 1514.527,A 0.000,B 0.000,C 90.000,E1 310.782} C_DIS
LIN {X 0.262,Y -390.610,Z 1514.495,A 0.000,B 0.000,C 90.000,E1 305.025} C_DIS
LIN {X 0.106,Y -391.104,Z 1514.493,A 0.000,B 0.000,C 90.000,E1 304.692} C_DIS
LIN {X 0.022,Y -391.648,Z 1514.489,A 0.000,B 0.000,C 90.000,E1 303.992} C_DIS
LIN {X -0.080,Y -396.825,Z 1514.459,A 0.000,B 0.000,C 90.000,E1 298.693} C_DIS
LIN {X -0.210,Y -397.120,Z 1514.457,A 0.000,B 0.000,C 90.000,E1 298.359} C_DIS
LIN {X -0.055,Y -401.597,Z 1514.426,A 0.000,B 0.000,C 90.000,E1 292.717} C_DIS
LIN {X 0.222,Y -404.659,Z 1514.395,A 0.000,B 0.000,C 90.000,E1 287.094} C_DIS
LIN {X -0.079,Y -404.735,Z 1514.391,A 0.000,B 0.000,C 90.000,E1 286.441} C_DIS
LIN {X 0.214,Y -406.099,Z 1514.364,A 0.000,B 0.000,C 90.000,E1 281.535} C_DIS
LIN {X -0.176,Y -406.094,Z 1514.362,A 0.000,B 0.000,C 90.000,E1 281.243} C_DIS
LIN {X -0.097,Y -405.680,Z 1514.333,A 0.000,B 0.000,C 90.000,E1 276.024} C_DIS
LIN {X -0.165,Y -405.058,Z 1514.328,A 0.000,B 0.000,C 90.000,E1 274.992} C_DIS
LIN {X -0.060,Y -403.497,Z 1514.304,A 0.000,B 0.000,C 90.000,E1 270.802} C_DIS
LIN {X -0.092,Y -403.288,Z 1514.302,A 0.000,B 0.000,C 90.000,E1 270.458} C_DIS
LIN {X 0.091,Y -398.931,Z 1514.271,A 0.000,B 0.000,C 90.000,E1 264.837} C_DIS
LIN {X -0.040,Y -393.108,Z 1514.242,A 0.000,B 0.000,C 90.000,E1 259.567} C_DIS
LIN {X -0.079,Y -392.835,Z 1514.240,A 0.000,B 0.000,C 90.000,E1 259.218} C_DIS
LIN {X 0.034,Y -385.993,Z 1514.212,A 0.000,B 0.000,C 90.000,E1 254.212} C_DIS
LIN {X -0.026,Y -385.267,Z 1514.208,A 0.000,B 0.000,C 90.000,E1 253.504} C_DIS
LIN {X -0.004,Y -384.768,Z 1514.206,A 0.000,B 0.000,C 90.000,E1 253.142} C_DIS
LIN {X 0.221,Y -377.973,Z 1514.182,A 0.000,B 0.000,C 90.000,E1 248.773} C_DIS
LIN {X -0.044,Y -376.233,Z 1514.174,A 0.000,B 0.000,C 90.000,E1 247.358} C_DIS
LIN {X 0.057,Y -374.944,Z 1514.170,A 0.000,B 0.000,C 90.000,E1 246.613} C_DIS
LIN {X -0.208,Y -368.417,Z 1514.148,A 0.000,B 0.000,C 90.000,E1 242.615} C_DIS
LIN {X 0.097,Y -366.047,Z 1514.137,A 0.000,B 0.000,C 90.000,E1 240.717} C_DIS
LIN {X 0.004,Y -359.196,Z 1514.115,A 0.000,B 0.000,C 90.000,E1 236.628} C_DIS
LIN {X 0.021,Y -355.842,Z 1514.100,A 0.000,B 0.000,C 90.000,E1 233.989} C_DIS
LIN {X -0.173,Y -348.793,Z 1514.075,A 0.000,B 0.000,C 90.000,E1 229.461} C_DIS
LIN {X -0.097,Y -346.185,Z 1514.062,A 0.000,B 0.000,C 90.000,E1 227.148} C_DIS
LIN {X -0.088,Y -345.065,Z 1514.058,A 0.000,B 0.000,C 90.000,E1 226.377} C_DIS
LIN {X 0.094,Y -338.586,Z 1514.030,A 0.000,B 0.000,C 90.000,E1 221.310} C_DIS
LIN {X 0.094,Y -336.840,Z 1514.019,A 0.000,B 0.000,C 90.000,E1 219.358} C_DIS
LIN {X 0.014,Y -330.861,Z 1513.988,A 0.000,B 0.000,C 90.000,E1 213.865} C_DIS
LIN {X 0.149,Y -329.296,Z 1513.975,A 0.000,B 0.000,C 90.000,E1 211.465} C_DIS
LIN {X -0.154,Y -324.669,Z 1513.942,A 0.000,B 0.000,C 90.000,E1 205.540} C_DIS
LIN {X 0.174,Y -323.837,Z 1513.928,A 0.000,B 0.000,C 90.000,E1 203.078} C_DIS
LIN {X -0.017,Y -321.124,Z 1513.881,A 0.000,B 0.000,C 90.000,E1 194.662} C_DIS
LIN {X 0.138,Y -320.932,Z 1513.877,A 0.000,B 0.000,C 90.000,E1 193.828} C_DIS
LIN {X -0.076,Y -321.562,Z 1513.832,A 0.000,B 0.000,C 90.000,E1 185.796} C_DIS
LIN {X -0.143,Y -324.415,Z 1513.790,A 0.000,B 0.000,C 90.000,E1 178.165} C_DIS
LIN {X -0.141,Y -325.376,Z 1513.783,A 0.000,B 0.000,C 90.000,E1 176.963} C_DIS
LIN {X -0.100,Y -329.112,Z 1513.750,A 0.000,B 0.000,C 90.000,E1 170.971} C_DIS
LIN {X 0.061,Y -334.260,Z 1513.726,A 0.000,B 0.000,C 90.000,E1 166.589} C_DIS
LIN {X 0.067,Y -335.488,Z 1513.719,A 0.000,B 0.000,C 90.000,E1 165.408} C_DIS
LIN {X 0.143,Y -340.932,Z 1513.695,A 0.000,B 0.000,C 90.000,E1 161.094} C_DIS
LIN {X -0.172,Y -342.138,Z 1513.691,A 0.000,B 0.000,C 90.000,E1 160.369} C_DIS
LIN {X -0.058,Y -347.939,Z 1513.667,A 0.000,B 0.000,C 90.000,E1 156.102} C_DIS
LIN {X -0.081,Y -354.259,Z 1513.648,A 0.000,B 0.000,C 90.000,E1 152.666} C_DIS
LIN {X -0.222,Y -361.406,Z 1513.625,A 0.000,B 0.000,C 90.000,E1 148.535} C_DIS
LIN {X 0.065,Y -368.758,Z 1513.606,A 0.000,B 0.000,C 90.000,E1 145.135} C_DIS
LIN {X -0.035,Y -376.505,Z 1513.585,A 0.000,B 0.000,C 90.000,E1 141.331} C_DIS
LIN {X -0.082,Y -536.155,Z 1513.585,A 0.000,B 0.000,C 90.000,E1 141.331} C_DIS
LIN {X -0.036,Y -538.532,Z 1513.585,A 0.000,B 0.000,C 90.000,E1 141.215} C_DIS
LIN {X 0.093,Y -539.565,Z 1513.584,A 0.000,B 0.000,C 90.000,E1 141.090} C_DIS
LIN {X 0.160,Y -541.369,Z 1513.582,A 0.000,B 0.000,C 90.000,E1 140.803} C_DIS
LIN {X 0.179,Y -542.775,Z 1513.581,A 0.000,B 0.000,C 90.000,E1 140.517} C_DIS
LIN {X -0.216,Y -543.918,Z 1513.579,A 0.000,B 0.000,C 90.000,E1 140.275} C_DIS
LIN {X -0.162,Y -545.719,Z 1513.576,A 0.000,B 0.000,C 90.000,E1 139.703} C_DIS
LIN {X -0.155,Y -547.124,Z 1513.573,A 0.000,B 0.000,C 90.000,E1 139.138} C_DIS
LIN {X -0.082,Y -548.221,Z 1513.570,A 0.000,B 0.000,C 90.000,E1 138.566} C_DIS
LIN {X -0.009,Y -549.486,Z 1513.565,A 0.000,B 0.000,C 90.000,E1 137.715} C_DIS
LIN {X 0.094,Y -550.995,Z 1513.559,A 0.000,B 0.000,C 90.000,E1 136.581} C_DIS
LIN {X -0.083,Y -552.977,Z 1513.550,A 0.000,B 0.000,C 90.000,E1 134.919} C_DIS
LIN {X 0.075,Y -554.092,Z 1513.543,A 0.000,B 0.000,C 90.000,E1 133.785} C_DIS
LIN {X -0.134,Y -555.119,Z 1513.537,A 0.000,B 0.000,C 90.000,E1 132.690} C_DIS
LIN {X -0.262,Y -556.204,Z 1513.529,A 0.000,B 0.000,C 90.000,E1 131.310} C_DIS
LIN {X 0.050,Y -557.156,Z 1513.522,A 0.000,B 0.000,C 90.000,E1 129.886} C_DIS
LIN {X 0.108,Y -558.357,Z 1513.511,A 0.000,B 0.000,C 90.000,E1 127.935} C_DIS
LIN {X -0.150,Y -559.246,Z 1513.502,A 0.000,B 0.000,C 90.000,E1 126.297} C_DIS
LIN {X -0.025,Y -559.677,Z 1513.494,A 0.000,B 0.000,C 90.000,E1 124.898} C_DIS
LIN {X 0.018,Y -559.879,Z 1513.488,A 0.000,B 0.000,C 90.000,E1 123.785} C_DIS
LIN {X -0.027,Y -559.871,Z 1513.483,A 0.000,B 0.000,C 90.000,E1 122.959} C_DIS
LIN {X -0.203,Y -559.970,Z 1513.468,A 0.000,B 0.000,C 90.000,E1 120.207} C_DIS
LIN {X -0.190,Y -560.255,Z 1513.460,A 0.000,B 0.000,C 90.000,E1 118.821} C_DIS
LIN {X 0.315,Y -560.540,Z 1513.452,A 0.000,B 0.000,C 90.000,E1 117.385} C_DIS
LIN {X -0.140,Y -560.896,Z 1513.443,A 0.000,B 0.000,C 90.000,E1 115.771} C_DIS
LIN {X -0.022,Y -561.285,Z 1513.432,A 0.000,B 0.000,C 90.000,E1 113.823} C_DIS
LIN {X -0.224,Y -561.500,Z 1513.425,A 0.000,B 0.000,C 90.000,E1 112.461} C_DIS
LIN {X -0.106,Y -561.815,Z 1513.416,A 0.000,B 0.000,C 90.000,E1 110.791} C_DIS
LIN {X 0.030,Y -562.110,Z 1513.408,A 0.000,B 0.000,C 90.000,E1 109.396} C_DIS
LIN {X -0.223,Y -562.374,Z 1513.399,A 0.000,B 0.000,C 90.000,E1 107.764} C_DIS
LIN {X 0.208,Y -562.822,Z 1513.388,A 0.000,B 0.000,C 90.000,E1 105.788} C_DIS
LIN {X 0.040,Y -563.173,Z 1513.380,A 0.000,B 0.000,C 90.000,E1 104.426} C_DIS
LIN {X 0.199,Y -563.690,Z 1513.370,A 0.000,B 0.000,C 90.000,E1 102.479} C_DIS
LIN {X -0.086,Y -564.203,Z 1513.362,A 0.000,B 0.000,C 90.000,E1 101.130} C_DIS
LIN {X 0.026,Y -565.135,Z 1513.350,A 0.000,B 0.000,C 90.000,E1 98.916} C_DIS
LIN {X -0.107,Y -565.902,Z 1513.339,A 0.000,B 0.000,C 90.000,E1 97.004} C_DIS
LIN {X -0.248,Y -566.998,Z 1513.327,A 0.000,B 0.000,C 90.000,E1 94.821} C_DIS
LIN {X -0.166,Y -567.649,Z 1513.319,A 0.000,B 0.000,C 90.000,E1 93.440} C_DIS
LIN {X 0.155,Y -568.667,Z 1513.308,A 0.000,B 0.000,C 90.000,E1 91.489} C_DIS
LIN {X -0.229,Y -569.555,Z 1513.299,A 0.000,B 0.000,C 90.000,E1 89.885} C_DIS
LIN {X 0.121,Y -570.640,Z 1513.289,A 0.000,B 0.000,C 90.000,E1 87.936} C_DIS
LIN {X 0.091,Y -571.849,Z 1513.276,A 0.000,B 0.000,C 90.000,E1 85.755} C_DIS
LIN {X 0.259,Y -572.640,Z 1513.269,A 0.000,B 0.000,C 90.000,E1 84.375} C_DIS
LIN {X -0.201,Y -574.057,Z 1513.257,A 0.000,B 0.000,C 90.000,E1 82.243} C_DIS
LIN {X -0.108,Y -575.400,Z 1513.246,A 0.000,B 0.000,C 90.000,E1 80.330} C_DIS
LIN {X 0.112,Y -576.815,Z 1513.236,A 0.000,B 0.000,C 90.000,E1 78.409} C_DIS
LIN {X -0.303,Y -578.069,Z 1513.227,A 0.000,B 0.000,C 90.000,E1 76.825} C_DIS
LIN {X -0.210,Y -579.046,Z 1513.219,A 0.000,B 0.000,C 90.000,E1 75.463} C_DIS
LIN {X 0.244,Y -579.826,Z 1513.213,A 0.000,B 0.000,C 90.000,E1 74.338} C_DIS
LIN {X -0.027,Y -580.671,Z 1513.206,A 0.000,B 0.000,C 90.000,E1 73.015} C_DIS
LIN {X 0.275,Y -581.530,Z 1513.198,A 0.000,B 0.000,C 90.000,E1 71.638} C_DIS
LIN {X 0.278,Y -582.643,Z 1513.188,A 0.000,B 0.000,C 90.000,E1 69.752} C_DIS
LIN {X -0.249,Y -583.677,Z 1513.177,A 0.000,B 0.000,C 90.000,E1 67.922} C_DIS
LIN {X -0.319,Y -584.735,Z 1513.167,A 0.000,B 0.000,C 90.000,E1 66.049} C_DIS
LIN {X -0.118,Y -585.793,Z 1513.156,A 0.000,B 0.000,C 90.000,E1 64.152} C_DIS
LIN {X -0.073,Y -586.545,Z 1513.150,A 0.000,B 0.000,C 90.000,E1 63.076} C_DIS
LIN {X 0.013,Y -587.744,Z 1513.141,A 0.000,B 0.000,C 90.000,E1 61.463} C_DIS
LIN {X 0.009,Y -588.709,Z 1513.134,A 0.000,B 0.000,C 90.000,E1 60.127} C_DIS
LIN {X -0.083,Y -589.808,Z 1513.125,A 0.000,B 0.000,C 90.000,E1 58.535} C_DIS
LIN {X -0.048,Y -590.760,Z 1513.118,A 0.000,B 0.000,C 90.000,E1 57.199} C_DIS
LIN {X 0.244,Y -592.139,Z 1513.107,A 0.000,B 0.000,C 90.000,E1 55.308} C_DIS
LIN {X -0.070,Y -592.756,Z 1513.102,A 0.000,B 0.000,C 90.000,E1 54.276} C_DIS
LIN {X -0.071,Y -593.479,Z 1513.093,A 0.000,B 0.000,C 90.000,E1 52.683} C_DIS
LIN {X -0.052,Y -594.195,Z 1513.084,A 0.000,B 0.000,C 90.000,E1 51.090} C_DIS
LIN {X 0.332,Y -595.114,Z 1513.072,A 0.000,B 0.000,C 90.000,E1 48.933} C_DIS
LIN {X -0.141,Y -595.348,Z 1513.066,A 0.000,B 0.000,C 90.000,E1 47.919} C_DIS
LIN {X 0.010,Y -595.290,Z 1513.059,A 0.000,B 0.000,C 90.000,E1 46.581} C_DIS
LIN {X 0.158,Y -595.070,Z 1513.052,A 0.000,B 0.000,C 90.000,E1 45.243} C_DIS
LIN {X 0.098,Y -594.569,Z 1513.046,A 0.000,B 0.000,C 90.000,E1 44.190} C_DIS
LIN {X 0.256,Y -594.078,Z 1513.041,A 0.000,B 0.000,C 90.000,E1 43.380} C_DIS
LIN {X -0.028,Y -592.871,Z 1513.034,A 0.000,B 0.000,C 90.000,E1 42.081} C_DIS
LIN {X 0.062,Y -591.532,Z 1513.026,A 0.000,B 0.000,C 90.000,E1 40.744} C_DIS
LIN {X 0.227,Y -590.593,Z 1513.022,A 0.000,B 0.000,C 90.000,E1 39.930} C_DIS
LIN {X -0.242,Y -589.122,Z 1513.016,A 0.000,B 0.000,C 90.000,E1 38.910} C_DIS
LIN {X -0.098,Y -587.722,Z 1513.012,A 0.000,B 0.000,C 90.000,E1 38.096} C_DIS
LIN {X 0.297,Y -586.557,Z 1513.009,A 0.000,B 0.000,C 90.000,E1 37.523} C_DIS
LIN {X -0.135,Y -584.997,Z 1513.006,A 0.000,B 0.000,C 90.000,E1 37.030} C_DIS
LIN {X -0.226,Y -582.943,Z 1513.003,A 0.000,B 0.000,C 90.000,E1 36.503} C_DIS
LIN {X -0.044,Y -581.688,Z 1513.001,A 0.000,B 0.000,C 90.000,E1 36.217} C_DIS
LIN {X 0.131,Y -580.120,Z 1513.000,A 0.000,B 0.000,C 90.000,E1 35.931} C_DIS
LIN {X 0.047,Y -579.167,Z 1512.999,A 0.000,B 0.000,C 90.000,E1 35.804} C_DIS
LIN {X 0.185,Y -577.386,Z 1512.998,A 0.000,B 0.000,C 90.000,E1 35.598} C_DIS
LIN {X 0.020,Y -575.970,Z 1512.997,A 0.000,B 0.000,C 90.000,E1 35.518} C_DIS
LIN {X 0.145,Y -574.933,Z 1512.997,A 0.000,B 0.000,C 90.000,E1 35.471} C_DIS
LIN {X 0.112,Y -574.611,Z 1512.997,A 0.000,B 0.000,C 90.000,E1 35.471} C_DIS
LIN {X 0.054,Y -399.641,Z 1512.997,A 0.000,B 0.000,C 90.000,E1 35.471} C_DIS
LIN {X 0.044,Y -393.864,Z 1512.977,A 0.000,B 0.000,C 90.000,E1 31.878} C_DIS
LIN {X -0.178,Y -386.451,Z 1512.953,A 0.000,B 0.000,C 90.000,E1 27.641} C_DIS
LIN {X -0.202,Y -382.757,Z 1512.938,A 0.000,B 0.000,C 90.000,E1 24.771} C_DIS
LIN {X 0.237,Y -376.075,Z 1512.911,A 0.000,B 0.000,C 90.000,E1 19.993} C_DIS
LIN {X 0.096,Y -373.610,Z 1512.897,A 0.000,B 0.000,C 90.000,E1 17.457} C_DIS
LIN {X 0.130,Y -368.014,Z 1512.869,A 0.000,B 0.000,C 90.000,E1 12.299} C_DIS
LIN {X 0.147,Y -366.575,Z 1512.856,A 0.000,B 0.000,C 90.000,E1 10.074} C_DIS
LIN {X 0.003,Y -366.302,Z 1512.854,A 0.000,B 0.000,C 90.000,E1 9.726} C_DIS
LIN {X -0.118,Y -361.702,Z 1512.821,A 0.000,B 0.000,C 90.000,E1 3.784} C_DIS
LIN {X -0.037,Y -360.909,Z 1512.802,A 0.000,B 0.000,C 90.000,E1 0.401} C_DIS
LIN {X 0.137,Y -360.684,Z 1512.799,A 0.000,B 0.000,C 90.000,E1 359.771} C_DIS
LIN {X -0.053,Y -359.426,Z 1512.770,A 0.000,B 0.000,C 90.000,E1 354.546} C_DIS
LIN {X 0.070,Y -358.890,Z 1512.759,A 0.000,B 0.000,C 90.000,E1 352.648} C_DIS
LIN {X -0.020,Y -359.563,Z 1512.726,A 0.000,B 0.000,C 90.000,E1 346.645} C_DIS
LIN {X 0.001,Y -361.801,Z 1512.684,A 0.000,B 0.000,C 90.000,E1 339.135} C_DIS
LIN {X -0.154,Y -362.053,Z 1512.680,A 0.000,B 0.000,C 90.000,E1 338.411} C_DIS
LIN {X 0.189,Y -365.980,Z 1512.643,A 0.000,B 0.000,C 90.000,E1 331.641} C_DIS
LIN {X 0.029,Y -366.387,Z 1512.639,A 0.000,B 0.000,C 90.000,E1 330.923} C_DIS
LIN {X -0.031,Y -371.355,Z 1512.604,A 0.000,B 0.000,C 90.000,E1 324.642} C_DIS
LIN {X -0.043,Y -371.766,Z 1512.602,A 0.000,B 0.000,C 90.000,E1 324.276} C_DIS
LIN {X 0.013,Y -377.358,Z 1512.567,A 0.000,B 0.000,C 90.000,E1 318.038} C_DIS
LIN {X 0.012,Y -378.235,Z 1512.563,A 0.000,B 0.000,C 90.000,E1 317.310} C_DIS
LIN {X 0.002,Y -383.940,Z 1512.531,A 0.000,B 0.000,C 90.000,E1 311.515} C_DIS
LIN {X 0.088,Y -384.893,Z 1512.527,A 0.000,B 0.000,C 90.000,E1 310.782} C_DIS
LIN {X 0.262,Y -390.610,Z 1512.495,A 0.000,B 0.000,C 90.000,E1 305.025} C_DIS
LIN {X 0.106,Y -391.104,Z 1512.493,A 0.000,B 0.000,C 90.000,E1 304.692} C_DIS
LIN {X 0.022,Y -391.648,Z 1512.489,A 0.000,B 0.000,C 90.000,E1 303.992} C_DIS
LIN {X -0.080,Y -396.825,Z 1512.459,A 0.000,B 0.000,C 90.000,E1 298.693} C_DIS
LIN {X -0.210,Y -397.120,Z 1512.457,A 0.000,B 0.000,C 90.000,E1 298.359} C_DIS
LIN {X -0.055,Y -401.597,Z 1512.426,A 0.000,B 0.000,C 90.000,E1 292.717} C_DIS
LIN {X 0.222,Y -404.659,Z 1512.395,A 0.000,B 0.000,C 90.000,E1 287.094} C_DIS
LIN {X -0.079,Y -404.735,Z 1512.391,A 0.000,B 0.000,C 90.000,E1 286.441} C_DIS
LIN {X 0.214,Y -406.099,Z 1512.364,A 0.000,B 0.000,C 90.000,E1 281.535} C_DIS
LIN {X -0.176,Y -406.094,Z 1512.362,A 0.000,B 0.000,C 90.000,E1 281.243} C_DIS
LIN {X -0.097,Y -405.680,Z 1512.333,A 0.000,B 0.000,C 90.000,E1 276.024} C_DIS
LIN {X -0.165,Y -405.058,Z 1512.328,A 0.000,B 0.000,C 90.000,E1 274.992} C_DIS
LIN {X -0.060,Y -403.497,Z 1512.304,A 0.000,B 0.000,C 90.000,E1 270.802} C_DIS
LIN {X -0.092,Y -403.288,Z 1512.302,A 0.000,B 0.000,C 90.000,E1 270.458} C_DIS
LIN {X 0.091,Y -398.931,Z 1512.271,A 0.000,B 0.000,C 90.000,E1 264.837} C_DIS
LIN {X -0.040,Y -393.108,Z 1512.242,A 0.000,B 0.000,C 90.000,E1 259.567} C_DIS
LIN {X -0.079,Y -392.835,Z 1512.240,A 0.000,B 0.000,C 90.000,E1 259.218} C_DIS
LIN {X 0.034,Y -385.993,Z 1512.212,A 0.000,B 0.000,C 90.000,E1 254.212} C_DIS
LIN {X -0.026,Y -385.267,Z 1512.208,A 0.000,B 0.000,C 90.000,E1 253.504} C_DIS
LIN {X -0.004,Y -384.768,Z 1512.206,A 0.000,B 0.000,C 90.000,E1 253.142} C_DIS
LIN {X 0.221,Y -377.973,Z 1512.182,A 0.000,B 0.000,C 90.000,E1 248.773} C_DIS
LIN {X -0.044,Y -376.233,Z 1512.174,A 0.000,B 0.000,C 90.000,E1 247.358} C_DIS
LIN {X 0.057,Y -374.944,Z 1512.170,A 0.000,B 0.000,C 90.000,E1 246.613} C_DIS
LIN {X -0.208,Y -368.417,Z 1512.148,A 0.000,B 0.000,C 90.000,E1 242.615} C_DIS
LIN {X 0.097,Y -366.047,Z 1512.137,A 0.000,B 0.000,C 90.000,E1 240.717} C_DIS
LIN {X 0.004,Y -359.196,Z 1512.115,A 0.000,B 0.000,C 90.000,E1 236.628} C_DIS
LIN {X 0.021,Y -355.842,Z 1512.100,A 0.000,B 0.000,C 90.000,E1 233.989} C_DIS
LIN {X -0.173,Y -348.793,Z 1512.075,A 0.000,B 0.000,C 90.000,E1 229.461} C_DIS
LIN {X -0.097,Y -346.185,Z 1512.062,A 0.000,B 0.000,C 90.000,E1 227.148} C_DIS
LIN {X -0.088,Y -345.065,Z 1512.058,A 0.000,B 0.000,C 90.000,E1 226.377} C_DIS
LIN {X 0.094,Y -338.586,Z 1512.030,A 0.000,B 0.000,C 90.000,E1 221.310} C_DIS
LIN {X 0.094,Y -336.840,Z 1512.019,A 0.000,B 0.000,C 90.000,E1 219.358} C_DIS
LIN {X 0.014,Y -330.861,Z 1511.988,A 0.000,B 0.000,C 90.000,E1 213.865} C_DIS
LIN {X 0.149,Y -329.296,Z 1511.975,A 0.000,B 0.000,C 90.000,E1 211.465} C_DIS
LIN {X -0.154,Y -324.669,Z 1511.942,A 0.000,B 0.000,C 90.000,E1 205.540} C_DIS
LIN {X 0.174,Y -323.837,Z 1511.928,A 0.000,B 0.000,C 90.000,E1 203.078} C_DIS
LIN {X -0.017,Y -321.124,Z 1511.881,A 0.000,B 0.000,C 90.000,E1 194.662} C_DIS
LIN {X 0.138,Y -320.932,Z 1511.877,A 0.000,B 0.000,C 90.000,E1 193.828} C_DIS
LIN {X -0.076,Y -321.562,Z 1511.832,A 0.000,B 0.000,C 90.000,E1 185.796} C_DIS
LIN {X -0.143,Y -324.415,Z 1511.790,A 0.000,B 0.000,C 90.000,E1 178.165} C_DIS
LIN {X -0.141,Y -325.376,Z 1511.783,A 0.000,B 0.000,C 90.000,E1 176.963} C_DIS
LIN {X -0.100,Y -329.112,Z 1511.750,A 0.000,B 0.000,C 90.000,E1 170.971} C_DIS
LIN {X 0.061,Y -334.260,Z 1511.726,A 0.000,B 0.000,C 90.000,E1 166.589} C_DIS
LIN {X 0.067,Y -335.488,Z 1511.719,A 0.000,B 0.000,C 90.000,E1 165.408} C_DIS
LIN {X 0.143,Y -340.932,Z 1511.695,A 0.000,B 0.000,C 90.000,E1 161.094} C_DIS
LIN {X -0.172,Y -342.138,Z 1511.691,A 0.000,B 0.000,C 90.000,E1 160.369} C_DIS
LIN {X -0.058,Y -347.939,Z 1511.667,A 0.000,B 0.000,C 90.000,E1 156.102} C_DIS
LIN {X -0.081,Y -354.259,Z 1511.648,A 0.000,B 0.000,C 90.000,E1 152.666} C_DIS
LIN {X -0.222,Y -361.406,Z 1511.625,A 0.000,B 0.000,C 90.000,E1 148.535} C_DIS
LIN {X 0.065,Y -368.758,Z 1511.606,A 0.000,B 0.000,C 90.000,E1 145.135} C_DIS
LIN {X -0.005,Y -374.751,Z 1511.590,A 0.000,B 0.000,C 90.000,E1 142.110} C_DIS
LIN {X -0.047,Y -535.352,Z 1511.589,A 0.000,B 0.000,C 90.000,E1 142.110} C_DIS
LIN {X -0.088,Y -535.577,Z 1511.589,A 0.000,B 0.000,C 90.000,E1 142.110} C_DIS
LIN {X -0.175,Y -537.781,Z 1511.589,A 0.000,B 0.000,C 90.000,E1 141.984} C_DIS
LIN {X 0.068,Y -538.949,Z 1511.588,A 0.000,B 0.000,C 90.000,E1 141.823} C_DIS
LIN {X 0.079,Y -540.724,Z 1511.586,A 0.000,B 0.000,C 90.000,E1 141.537} C_DIS
LIN {X 0.097,Y -542.106,Z 1511.585,A 0.000,B 0.000,C 90.000,E1 141.251} C_DIS
LIN {X 0.120,Y -543.207,Z 1511.583,A 0.000,B 0.000,C 90.000,E1 140.964} C_DIS
LIN {X -0.249,Y -545.026,Z 1511.580,A 0.000,B 0.000,C 90.000,E1 140.436} C_DIS
LIN {X 0.166,Y -546.410,Z 1511.577,A 0.000,B 0.000,C 90.000,E1 139.828} C_DIS
LIN {X -0.176,Y -547.514,Z 1511.574,A 0.000,B 0.000,C 90.000,E1 139.299} C_DIS
LIN {X -0.108,Y -548.829,Z 1511.569,A 0.000,B 0.000,C 90.000,E1 138.447} C_DIS
LIN {X 0.020,Y -550.460,Z 1511.563,A 0.000,B 0.000,C 90.000,E1 137.310} C_DIS
LIN {X -0.240,Y -551.836,Z 1511.557,A 0.000,B 0.000,C 90.000,E1 136.215} C_DIS
LIN {X -0.060,Y -553.445,Z 1511.549,A 0.000,B 0.000,C 90.000,E1 134.798} C_DIS
LIN {X -0.284,Y -554.526,Z 1511.543,A 0.000,B 0.000,C 90.000,E1 133.704} C_DIS
LIN {X 0.296,Y -555.496,Z 1511.536,A 0.000,B 0.000,C 90.000,E1 132.528} C_DIS
LIN {X 0.172,Y -556.551,Z 1511.529,A 0.000,B 0.000,C 90.000,E1 131.148} C_DIS
LIN {X 0.061,Y -557.481,Z 1511.521,A 0.000,B 0.000,C 90.000,E1 129.769} C_DIS
LIN {X 0.208,Y -558.650,Z 1511.510,A 0.000,B 0.000,C 90.000,E1 127.810} C_DIS
LIN {X -0.129,Y -559.368,Z 1511.503,A 0.000,B 0.000,C 90.000,E1 126.457} C_DIS
LIN {X 0.325,Y -559.790,Z 1511.495,A 0.000,B 0.000,C 90.000,E1 125.025} C_DIS
LIN {X 0.367,Y -560.011,Z 1511.489,A 0.000,B 0.000,C 90.000,E1 123.913} C_DIS
LIN {X 0.103,Y -559.959,Z 1511.483,A 0.000,B 0.000,C 90.000,E1 122.832} C_DIS
LIN {X 0.008,Y -560.143,Z 1511.466,A 0.000,B 0.000,C 90.000,E1 119.795} C_DIS
LIN {X -0.187,Y -560.469,Z 1511.456,A 0.000,B 0.000,C 90.000,E1 118.153} C_DIS
LIN {X -0.037,Y -560.936,Z 1511.444,A 0.000,B 0.000,C 90.000,E1 115.924} C_DIS
LIN {X 0.327,Y -561.304,Z 1511.433,A 0.000,B 0.000,C 90.000,E1 113.951} C_DIS
LIN {X -0.189,Y -561.504,Z 1511.427,A 0.000,B 0.000,C 90.000,E1 112.898} C_DIS
LIN {X 0.249,Y -561.867,Z 1511.416,A 0.000,B 0.000,C 90.000,E1 110.918} C_DIS
LIN {X 0.174,Y -562.217,Z 1511.407,A 0.000,B 0.000,C 90.000,E1 109.268} C_DIS
LIN {X 0.060,Y -562.545,Z 1511.396,A 0.000,B 0.000,C 90.000,E1 107.347} C_DIS
LIN {X 0.041,Y -562.883,Z 1511.389,A 0.000,B 0.000,C 90.000,E1 105.969} C_DIS
LIN {X 0.174,Y -563.323,Z 1511.380,A 0.000,B 0.000,C 90.000,E1 104.300} C_DIS
LIN {X -0.224,Y -563.854,Z 1511.369,A 0.000,B 0.000,C 90.000,E1 102.411} C_DIS
LIN {X 0.037,Y -564.362,Z 1511.361,A 0.000,B 0.000,C 90.000,E1 101.007} C_DIS
LIN {X 0.053,Y -565.324,Z 1511.349,A 0.000,B 0.000,C 90.000,E1 98.803} C_DIS
LIN {X -0.071,Y -566.090,Z 1511.338,A 0.000,B 0.000,C 90.000,E1 96.891} C_DIS
LIN {X -0.154,Y -567.207,Z 1511.326,A 0.000,B 0.000,C 90.000,E1 94.702} C_DIS
LIN {X 0.035,Y -568.016,Z 1511.317,A 0.000,B 0.000,C 90.000,E1 93.037} C_DIS
LIN {X 0.215,Y -568.931,Z 1511.308,A 0.000,B 0.000,C 90.000,E1 91.375} C_DIS
LIN {X 0.149,Y -569.511,Z 1511.302,A 0.000,B 0.000,C 90.000,E1 90.286} C_DIS
LIN {X -0.086,Y -570.614,Z 1511.291,A 0.000,B 0.000,C 90.000,E1 88.396} C_DIS
LIN {X -0.113,Y -571.245,Z 1511.285,A 0.000,B 0.000,C 90.000,E1 87.306} C_DIS
LIN {X -0.272,Y -572.384,Z 1511.274,A 0.000,B 0.000,C 90.000,E1 85.412} C_DIS
LIN {X -0.102,Y -573.134,Z 1511.267,A 0.000,B 0.000,C 90.000,E1 84.033} C_DIS
LIN {X -0.232,Y -574.246,Z 1511.258,A 0.000,B 0.000,C 90.000,E1 82.413} C_DIS
LIN {X -0.125,Y -575.590,Z 1511.247,A 0.000,B 0.000,C 90.000,E1 80.500} C_DIS
LIN {X -0.242,Y -577.224,Z 1511.235,A 0.000,B 0.000,C 90.000,E1 78.342} C_DIS
LIN {X -0.073,Y -578.487,Z 1511.226,A 0.000,B 0.000,C 90.000,E1 76.700} C_DIS
LIN {X 0.252,Y -579.617,Z 1511.217,A 0.000,B 0.000,C 90.000,E1 75.046} C_DIS
LIN {X 0.157,Y -580.390,Z 1511.211,A 0.000,B 0.000,C 90.000,E1 73.976} C_DIS
LIN {X 0.069,Y -581.067,Z 1511.205,A 0.000,B 0.000,C 90.000,E1 72.906} C_DIS
LIN {X -0.183,Y -581.898,Z 1511.198,A 0.000,B 0.000,C 90.000,E1 71.583} C_DIS
LIN {X 0.169,Y -582.845,Z 1511.189,A 0.000,B 0.000,C 90.000,E1 69.934} C_DIS
LIN {X -0.349,Y -583.871,Z 1511.178,A 0.000,B 0.000,C 90.000,E1 68.103} C_DIS
LIN {X 0.125,Y -584.926,Z 1511.168,A 0.000,B 0.000,C 90.000,E1 66.177} C_DIS
LIN {X -0.080,Y -585.859,Z 1511.159,A 0.000,B 0.000,C 90.000,E1 64.588} C_DIS
LIN {X 0.144,Y -587.090,Z 1511.148,A 0.000,B 0.000,C 90.000,E1 62.692} C_DIS
LIN {X -0.161,Y -588.142,Z 1511.141,A 0.000,B 0.000,C 90.000,E1 61.385} C_DIS
LIN {X -0.153,Y -589.083,Z 1511.134,A 0.000,B 0.000,C 90.000,E1 60.049} C_DIS
LIN {X -0.231,Y -590.206,Z 1511.125,A 0.000,B 0.000,C 90.000,E1 58.456} C_DIS
LIN {X -0.068,Y -591.009,Z 1511.119,A 0.000,B 0.000,C 90.000,E1 57.375} C_DIS
LIN {X -0.091,Y -592.359,Z 1511.108,A 0.000,B 0.000,C 90.000,E1 55.515} C_DIS
LIN {X 0.211,Y -592.888,Z 1511.104,A 0.000,B 0.000,C 90.000,E1 54.689} C_DIS
LIN {X 0.252,Y -593.389,Z 1511.098,A 0.000,B 0.000,C 90.000,E1 53.623} C_DIS
LIN {X 0.048,Y -593.977,Z 1511.091,A 0.000,B 0.000,C 90.000,E1 52.316} C_DIS
LIN {X -0.143,Y -594.573,Z 1511.083,A 0.000,B 0.000,C 90.000,E1 51.009} C_DIS
LIN {X 0.035,Y -595.385,Z 1511.073,A 0.000,B 0.000,C 90.000,E1 49.138} C_DIS
LIN {X 0.025,Y -595.573,Z 1511.070,A 0.000,B 0.000,C 90.000,E1 48.609} C_DIS
LIN {X -0.213,Y -595.703,Z 1511.066,A 0.000,B 0.000,C 90.000,E1 47.838} C_DIS
LIN {X 0.169,Y -595.687,Z 1511.060,A 0.000,B 0.000,C 90.000,E1 46.743} C_DIS
LIN {X 0.324,Y -595.486,Z 1511.052,A 0.000,B 0.000,C 90.000,E1 45.405} C_DIS
LIN {X 0.071,Y -595.213,Z 1511.048,A 0.000,B 0.000,C 90.000,E1 44.636} C_DIS
LIN {X 0.206,Y -594.398,Z 1511.041,A 0.000,B 0.000,C 90.000,E1 43.299} C_DIS
LIN {X -0.072,Y -593.210,Z 1511.033,A 0.000,B 0.000,C 90.000,E1 42.000} C_DIS
LIN {X 0.022,Y -591.865,Z 1511.026,A 0.000,B 0.000,C 90.000,E1 40.663} C_DIS
LIN {X 0.190,Y -590.898,Z 1511.021,A 0.000,B 0.000,C 90.000,E1 39.850} C_DIS
LIN {X -0.276,Y -589.398,Z 1511.016,A 0.000,B 0.000,C 90.000,E1 38.830} C_DIS
LIN {X 0.131,Y -588.487,Z 1511.013,A 0.000,B 0.000,C 90.000,E1 38.257} C_DIS
LIN {X 0.266,Y -586.960,Z 1511.008,A 0.000,B 0.000,C 90.000,E1 37.443} C_DIS
LIN {X -0.006,Y -586.404,Z 1511.007,A 0.000,B 0.000,C 90.000,E1 37.202} C_DIS
LIN {X 0.216,Y -584.144,Z 1511.002,A 0.000,B 0.000,C 90.000,E1 36.377} C_DIS
LIN {X -0.068,Y -583.179,Z 1511.001,A 0.000,B 0.000,C 90.000,E1 36.137} C_DIS
LIN {X 0.032,Y -581.466,Z 1510.999,A 0.000,B 0.000,C 90.000,E1 35.724} C_DIS
LIN {X 0.124,Y -579.294,Z 1510.996,A 0.000,B 0.000,C 90.000,E1 35.311} C_DIS
LIN {X 0.041,Y -578.413,Z 1510.995,A 0.000,B 0.000,C 90.000,E1 35.185} C_DIS
LIN {X -0.064,Y -576.606,Z 1510.994,A 0.000,B 0.000,C 90.000,E1 34.978} C_DIS
LIN {X -0.071,Y -575.207,Z 1510.994,A 0.000,B 0.000,C 90.000,E1 34.865} C_DIS
LIN {X -0.147,Y -574.076,Z 1510.993,A 0.000,B 0.000,C 90.000,E1 34.818} C_DIS
LIN {X -0.301,Y -573.298,Z 1510.993,A 0.000,B 0.000,C 90.000,E1 34.818} C_DIS
LIN {X 0.083,Y -398.385,Z 1510.993,A 0.000,B 0.000,C 90.000,E1 34.771} C_DIS
LIN {X -0.020,Y -393.729,Z 1510.977,A 0.000,B 0.000,C 90.000,E1 31.799} C_DIS
LIN {X 0.084,Y -386.321,Z 1510.953,A 0.000,B 0.000,C 90.000,E1 27.513} C_DIS
LIN {X -0.105,Y -383.088,Z 1510.939,A 0.000,B 0.000,C 90.000,E1 25.027} C_DIS
LIN {X 0.053,Y -381.994,Z 1510.935,A 0.000,B 0.000,C 90.000,E1 24.283} C_DIS
LIN {X -0.022,Y -375.578,Z 1510.909,A 0.000,B 0.000,C 90.000,E1 19.577} C_DIS
LIN {X -0.142,Y -373.495,Z 1510.897,A 0.000,B 0.000,C 90.000,E1 17.402} C_DIS
LIN {X -0.103,Y -367.942,Z 1510.868,A 0.000,B 0.000,C 90.000,E1 12.243} C_DIS
LIN {X -0.083,Y -366.528,Z 1510.856,A 0.000,B 0.000,C 90.000,E1 10.018} C_DIS
LIN {X 0.060,Y -365.034,Z 1510.847,A 0.000,B 0.000,C 90.000,E1 8.511} C_DIS
LIN {X 0.155,Y -361.083,Z 1510.810,A 0.000,B 0.000,C 90.000,E1 1.776} C_DIS
LIN {X 0.096,Y -360.905,Z 1510.802,A 0.000,B 0.000,C 90.000,E1 0.286} C_DIS
LIN {X -0.053,Y -359.426,Z 1510.770,A 0.000,B 0.000,C 90.000,E1 354.546} C_DIS
LIN {X 0.070,Y -358.890,Z 1510.759,A 0.000,B 0.000,C 90.000,E1 352.648} C_DIS
LIN {X -0.020,Y -359.563,Z 1510.726,A 0.000,B 0.000,C 90.000,E1 346.645} C_DIS
LIN {X 0.001,Y -361.801,Z 1510.684,A 0.000,B 0.000,C 90.000,E1 339.135} C_DIS
LIN {X -0.154,Y -362.053,Z 1510.680,A 0.000,B 0.000,C 90.000,E1 338.411} C_DIS
LIN {X 0.189,Y -365.980,Z 1510.643,A 0.000,B 0.000,C 90.000,E1 331.641} C_DIS
LIN {X 0.029,Y -366.387,Z 1510.639,A 0.000,B 0.000,C 90.000,E1 330.923} C_DIS
LIN {X -0.031,Y -371.355,Z 1510.604,A 0.000,B 0.000,C 90.000,E1 324.642} C_DIS
LIN {X -0.043,Y -371.766,Z 1510.602,A 0.000,B 0.000,C 90.000,E1 324.276} C_DIS
LIN {X 0.013,Y -377.358,Z 1510.567,A 0.000,B 0.000,C 90.000,E1 318.038} C_DIS
LIN {X 0.012,Y -378.235,Z 1510.563,A 0.000,B 0.000,C 90.000,E1 317.310} C_DIS
LIN {X 0.002,Y -383.940,Z 1510.531,A 0.000,B 0.000,C 90.000,E1 311.515} C_DIS
LIN {X 0.088,Y -384.893,Z 1510.527,A 0.000,B 0.000,C 90.000,E1 310.782} C_DIS
LIN {X 0.262,Y -390.610,Z 1510.495,A 0.000,B 0.000,C 90.000,E1 305.025} C_DIS
LIN {X 0.106,Y -391.104,Z 1510.493,A 0.000,B 0.000,C 90.000,E1 304.692} C_DIS
LIN {X 0.022,Y -391.648,Z 1510.489,A 0.000,B 0.000,C 90.000,E1 303.992} C_DIS
LIN {X -0.080,Y -396.825,Z 1510.459,A 0.000,B 0.000,C 90.000,E1 298.693} C_DIS
LIN {X -0.210,Y -397.120,Z 1510.457,A 0.000,B 0.000,C 90.000,E1 298.359} C_DIS
LIN {X -0.055,Y -401.597,Z 1510.426,A 0.000,B 0.000,C 90.000,E1 292.717} C_DIS
LIN {X 0.222,Y -404.659,Z 1510.395,A 0.000,B 0.000,C 90.000,E1 287.094} C_DIS
LIN {X -0.079,Y -404.735,Z 1510.391,A 0.000,B 0.000,C 90.000,E1 286.441} C_DIS
LIN {X 0.214,Y -406.099,Z 1510.364,A 0.000,B 0.000,C 90.000,E1 281.535} C_DIS
LIN {X -0.176,Y -406.094,Z 1510.362,A 0.000,B 0.000,C 90.000,E1 281.243} C_DIS
LIN {X -0.097,Y -405.680,Z 1510.333,A 0.000,B 0.000,C 90.000,E1 276.024} C_DIS
LIN {X -0.165,Y -405.058,Z 1510.328,A 0.000,B 0.000,C 90.000,E1 274.992} C_DIS
LIN {X -0.060,Y -403.497,Z 1510.304,A 0.000,B 0.000,C 90.000,E1 270.802} C_DIS
LIN {X -0.092,Y -403.288,Z 1510.302,A 0.000,B 0.000,C 90.000,E1 270.458} C_DIS
LIN {X 0.091,Y -398.931,Z 1510.271,A 0.000,B 0.000,C 90.000,E1 264.837} C_DIS
LIN {X -0.040,Y -393.108,Z 1510.242,A 0.000,B 0.000,C 90.000,E1 259.567} C_DIS
LIN {X -0.079,Y -392.835,Z 1510.240,A 0.000,B 0.000,C 90.000,E1 259.218} C_DIS
LIN {X 0.034,Y -385.993,Z 1510.212,A 0.000,B 0.000,C 90.000,E1 254.212} C_DIS
LIN {X -0.026,Y -385.267,Z 1510.208,A 0.000,B 0.000,C 90.000,E1 253.504} C_DIS
LIN {X -0.004,Y -384.768,Z 1510.206,A 0.000,B 0.000,C 90.000,E1 253.142} C_DIS
LIN {X 0.221,Y -377.973,Z 1510.182,A 0.000,B 0.000,C 90.000,E1 248.773} C_DIS
LIN {X -0.044,Y -376.233,Z 1510.174,A 0.000,B 0.000,C 90.000,E1 247.358} C_DIS
LIN {X 0.057,Y -374.944,Z 1510.170,A 0.000,B 0.000,C 90.000,E1 246.613} C_DIS
LIN {X -0.208,Y -368.417,Z 1510.148,A 0.000,B 0.000,C 90.000,E1 242.615} C_DIS
LIN {X 0.097,Y -366.047,Z 1510.137,A 0.000,B 0.000,C 90.000,E1 240.717} C_DIS
LIN {X 0.004,Y -359.196,Z 1510.115,A 0.000,B 0.000,C 90.000,E1 236.628} C_DIS
LIN {X 0.021,Y -355.842,Z 1510.100,A 0.000,B 0.000,C 90.000,E1 233.989} C_DIS
LIN {X -0.173,Y -348.793,Z 1510.075,A 0.000,B 0.000,C 90.000,E1 229.461} C_DIS
LIN {X -0.097,Y -346.185,Z 1510.062,A 0.000,B 0.000,C 90.000,E1 227.148} C_DIS
LIN {X -0.088,Y -345.065,Z 1510.058,A 0.000,B 0.000,C 90.000,E1 226.377} C_DIS
LIN {X 0.094,Y -338.586,Z 1510.030,A 0.000,B 0.000,C 90.000,E1 221.310} C_DIS
LIN {X 0.094,Y -336.840,Z 1510.019,A 0.000,B 0.000,C 90.000,E1 219.358} C_DIS
LIN {X 0.014,Y -330.861,Z 1509.988,A 0.000,B 0.000,C 90.000,E1 213.865} C_DIS
LIN {X 0.149,Y -329.296,Z 1509.975,A 0.000,B 0.000,C 90.000,E1 211.465} C_DIS
LIN {X -0.154,Y -324.669,Z 1509.942,A 0.000,B 0.000,C 90.000,E1 205.540} C_DIS
LIN {X 0.174,Y -323.837,Z 1509.928,A 0.000,B 0.000,C 90.000,E1 203.078} C_DIS
LIN {X -0.017,Y -321.124,Z 1509.881,A 0.000,B 0.000,C 90.000,E1 194.662} C_DIS
LIN {X 0.138,Y -320.932,Z 1509.877,A 0.000,B 0.000,C 90.000,E1 193.828} C_DIS
LIN {X -0.076,Y -321.562,Z 1509.832,A 0.000,B 0.000,C 90.000,E1 185.796} C_DIS
LIN {X -0.143,Y -324.415,Z 1509.790,A 0.000,B 0.000,C 90.000,E1 178.165} C_DIS
LIN {X -0.141,Y -325.376,Z 1509.783,A 0.000,B 0.000,C 90.000,E1 176.963} C_DIS
LIN {X -0.100,Y -329.112,Z 1509.750,A 0.000,B 0.000,C 90.000,E1 170.971} C_DIS
LIN {X 0.061,Y -334.260,Z 1509.726,A 0.000,B 0.000,C 90.000,E1 166.589} C_DIS
LIN {X 0.067,Y -335.488,Z 1509.719,A 0.000,B 0.000,C 90.000,E1 165.408} C_DIS
LIN {X 0.143,Y -340.932,Z 1509.695,A 0.000,B 0.000,C 90.000,E1 161.094} C_DIS
LIN {X -0.172,Y -342.138,Z 1509.691,A 0.000,B 0.000,C 90.000,E1 160.369} C_DIS
LIN {X -0.058,Y -347.939,Z 1509.667,A 0.000,B 0.000,C 90.000,E1 156.102} C_DIS
LIN {X -0.081,Y -354.259,Z 1509.648,A 0.000,B 0.000,C 90.000,E1 152.666} C_DIS
LIN {X -0.222,Y -361.406,Z 1509.625,A 0.000,B 0.000,C 90.000,E1 148.535} C_DIS
LIN {X 0.065,Y -368.758,Z 1509.606,A 0.000,B 0.000,C 90.000,E1 145.135} C_DIS
LIN {X -0.032,Y -373.101,Z 1509.594,A 0.000,B 0.000,C 90.000,E1 142.889} C_DIS
LIN {X -0.090,Y -533.923,Z 1509.594,A 0.000,B 0.000,C 90.000,E1 142.889} C_DIS
LIN {X 0.247,Y -534.508,Z 1509.594,A 0.000,B 0.000,C 90.000,E1 142.844} C_DIS
LIN {X -0.007,Y -536.850,Z 1509.593,A 0.000,B 0.000,C 90.000,E1 142.718} C_DIS
LIN {X 0.063,Y -538.117,Z 1509.592,A 0.000,B 0.000,C 90.000,E1 142.557} C_DIS
LIN {X 0.070,Y -539.867,Z 1509.590,A 0.000,B 0.000,C 90.000,E1 142.271} C_DIS
LIN {X 0.086,Y -541.243,Z 1509.589,A 0.000,B 0.000,C 90.000,E1 141.984} C_DIS
LIN {X 0.107,Y -542.373,Z 1509.587,A 0.000,B 0.000,C 90.000,E1 141.698} C_DIS
LIN {X -0.269,Y -544.235,Z 1509.584,A 0.000,B 0.000,C 90.000,E1 141.170} C_DIS
LIN {X 0.174,Y -546.240,Z 1509.579,A 0.000,B 0.000,C 90.000,E1 140.275} C_DIS
LIN {X -0.091,Y -548.111,Z 1509.573,A 0.000,B 0.000,C 90.000,E1 139.175} C_DIS
LIN {X 0.021,Y -549.785,Z 1509.567,A 0.000,B 0.000,C 90.000,E1 138.038} C_DIS
LIN {X 0.124,Y -551.323,Z 1509.561,A 0.000,B 0.000,C 90.000,E1 136.905} C_DIS
LIN {X -0.122,Y -552.640,Z 1509.554,A 0.000,B 0.000,C 90.000,E1 135.810} C_DIS
LIN {X 0.034,Y -553.883,Z 1509.548,A 0.000,B 0.000,C 90.000,E1 134.676} C_DIS
LIN {X 0.205,Y -554.947,Z 1509.542,A 0.000,B 0.000,C 90.000,E1 133.542} C_DIS
LIN {X 0.071,Y -556.073,Z 1509.534,A 0.000,B 0.000,C 90.000,E1 132.162} C_DIS
LIN {X -0.038,Y -557.089,Z 1509.527,A 0.000,B 0.000,C 90.000,E1 130.782} C_DIS
LIN {X -0.140,Y -557.948,Z 1509.519,A 0.000,B 0.000,C 90.000,E1 129.402} C_DIS
LIN {X -0.069,Y -558.941,Z 1509.510,A 0.000,B 0.000,C 90.000,E1 127.729} C_DIS
LIN {X 0.288,Y -559.487,Z 1509.503,A 0.000,B 0.000,C 90.000,E1 126.583} C_DIS
LIN {X -0.129,Y -559.853,Z 1509.497,A 0.000,B 0.000,C 90.000,E1 125.518} C_DIS
LIN {X 0.003,Y -560.107,Z 1509.490,A 0.000,B 0.000,C 90.000,E1 124.119} C_DIS
LIN {X 0.046,Y -560.092,Z 1509.483,A 0.000,B 0.000,C 90.000,E1 123.007} C_DIS
LIN {X -0.137,Y -560.119,Z 1509.468,A 0.000,B 0.000,C 90.000,E1 120.256} C_DIS
LIN {X -0.128,Y -560.404,Z 1509.460,A 0.000,B 0.000,C 90.000,E1 118.871} C_DIS
LIN {X -0.085,Y -560.683,Z 1509.451,A 0.000,B 0.000,C 90.000,E1 117.206} C_DIS
LIN {X 0.174,Y -561.001,Z 1509.443,A 0.000,B 0.000,C 90.000,E1 115.796} C_DIS
LIN {X -0.202,Y -561.389,Z 1509.433,A 0.000,B 0.000,C 90.000,E1 113.898} C_DIS
LIN {X -0.180,Y -561.615,Z 1509.425,A 0.000,B 0.000,C 90.000,E1 112.514} C_DIS
LIN {X 0.144,Y -561.948,Z 1509.417,A 0.000,B 0.000,C 90.000,E1 111.099} C_DIS
LIN {X -0.333,Y -562.324,Z 1509.407,A 0.000,B 0.000,C 90.000,E1 109.214} C_DIS
LIN {X -0.128,Y -562.734,Z 1509.394,A 0.000,B 0.000,C 90.000,E1 106.985} C_DIS
LIN {X 0.094,Y -562.947,Z 1509.390,A 0.000,B 0.000,C 90.000,E1 106.134} C_DIS
LIN {X 0.075,Y -563.414,Z 1509.380,A 0.000,B 0.000,C 90.000,E1 104.481} C_DIS
LIN {X 0.235,Y -563.921,Z 1509.370,A 0.000,B 0.000,C 90.000,E1 102.535} C_DIS
LIN {X 0.117,Y -564.520,Z 1509.361,A 0.000,B 0.000,C 90.000,E1 100.894} C_DIS
LIN {X 0.067,Y -565.361,Z 1509.350,A 0.000,B 0.000,C 90.000,E1 98.973} C_DIS
LIN {X -0.132,Y -566.155,Z 1509.339,A 0.000,B 0.000,C 90.000,E1 97.068} C_DIS
LIN {X -0.043,Y -567.407,Z 1509.326,A 0.000,B 0.000,C 90.000,E1 94.588} C_DIS
LIN {X 0.154,Y -568.263,Z 1509.316,A 0.000,B 0.000,C 90.000,E1 92.922} C_DIS
LIN {X -0.229,Y -569.189,Z 1509.307,A 0.000,B 0.000,C 90.000,E1 91.318} C_DIS
LIN {X 0.151,Y -569.656,Z 1509.303,A 0.000,B 0.000,C 90.000,E1 90.458} C_DIS
LIN {X -0.081,Y -570.744,Z 1509.292,A 0.000,B 0.000,C 90.000,E1 88.568} C_DIS
LIN {X -0.106,Y -571.425,Z 1509.286,A 0.000,B 0.000,C 90.000,E1 87.478} C_DIS
LIN {X -0.126,Y -572.733,Z 1509.274,A 0.000,B 0.000,C 90.000,E1 85.298} C_DIS
LIN {X 0.235,Y -573.648,Z 1509.265,A 0.000,B 0.000,C 90.000,E1 83.628} C_DIS
LIN {X 0.120,Y -574.810,Z 1509.256,A 0.000,B 0.000,C 90.000,E1 82.008} C_DIS
LIN {X 0.032,Y -575.966,Z 1509.247,A 0.000,B 0.000,C 90.000,E1 80.387} C_DIS
LIN {X -0.082,Y -577.620,Z 1509.235,A 0.000,B 0.000,C 90.000,E1 78.229} C_DIS
LIN {X 0.088,Y -578.876,Z 1509.226,A 0.000,B 0.000,C 90.000,E1 76.589} C_DIS
LIN {X 0.071,Y -580.200,Z 1509.215,A 0.000,B 0.000,C 90.000,E1 74.700} C_DIS
LIN {X -0.240,Y -580.783,Z 1509.211,A 0.000,B 0.000,C 90.000,E1 73.921} C_DIS
LIN {X -0.154,Y -581.444,Z 1509.205,A 0.000,B 0.000,C 90.000,E1 72.834} C_DIS
LIN {X 0.161,Y -582.244,Z 1509.197,A 0.000,B 0.000,C 90.000,E1 71.456} C_DIS
LIN {X -0.222,Y -583.193,Z 1509.188,A 0.000,B 0.000,C 90.000,E1 69.880} C_DIS
LIN {X 0.020,Y -584.212,Z 1509.178,A 0.000,B 0.000,C 90.000,E1 67.975} C_DIS
LIN {X -0.029,Y -585.260,Z 1509.167,A 0.000,B 0.000,C 90.000,E1 66.102} C_DIS
LIN {X 0.058,Y -586.231,Z 1509.158,A 0.000,B 0.000,C 90.000,E1 64.485} C_DIS
LIN {X 0.137,Y -587.326,Z 1509.149,A 0.000,B 0.000,C 90.000,E1 62.871} C_DIS
LIN {X 0.245,Y -588.512,Z 1509.141,A 0.000,B 0.000,C 90.000,E1 61.257} C_DIS
